(* Logix 5000 project; controller PRU vendor 1 type 14 code 107 rev 20.13; software revision 20.01; part 4 of 17 *)
(* tags used below, declared in another part *)
   AFI : BOOL;
   AlarmMaster : DINT;
   ALL_AUTO_IOK : BOOL;   // All equipment is in Auto Mode.
   ALL_DRIVES_ARE_CMD_FWD : BOOL;
   ALL_DRIVES_ARE_READY : BOOL;
   ALL_SHUTDOWN_FAULTS_IOK : BOOL;
   AUTO_FWD_CMD_GON : BOOL;
   CHANGING_TOTE_2 : BOOL;
   CHANGING_TOTE_3 : BOOL;
   CHANGING_TOTE_4 : BOOL;
   CHANGING_TOTE_5 : BOOL;
   COOLSCREW : VFD;
   DRYER : DUAL_SCREW;
   DRYER_FWD_MODE : BOOL;
   FAULTS_FA4_IOK : BOOL;   // HI TEMP FAULTS ARE OK.
   FAULTS_FA5_IOK : BOOL;
   FWD_CMD_BON : TIMER;

        [3601] := 267.2754, [3602] := 267.45117, [3603] := 267.36328, [3604] := 267.80273, [3605] := 267.71484, [3606] := 267.53906, [3607] := 267.62695, [3608] := 268.50586, [3609] := 268.41797, [3610] := 268.2422, [3611] := 268.33008, [3612] := 267.89062, [3613] := 267.97852, [3614] := 268.1543, [3615] := 268.0664, [3616] := 264.375, [3617] := 264.4629, [3618] := 264.63867, [3619] := 264.55078, [3620] := 264.99023, [3621] := 264.90234, [3622] := 264.72656, [3623] := 264.81445, [3624] := 265.69336, [3625] := 265.60547, [3626] := 265.4297, [3627] := 265.51758, [3628] := 265.07812, [3629] := 265.16602, [3630] := 265.3418, [3631] := 265.2539, [3632] := 267.0996, [3633] := 267.01172, [3634] := 266.83594, [3635] := 266.92383, [3636] := 266.48438, [3637] := 266.57227, [3638] := 266.74805, [3639] := 266.66016, [3640] := 265.78125, [3641] := 265.86914, [3642] := 266.04492, [3643] := 265.95703, [3644] := 266.39648, [3645] := 266.3086, [3646] := 266.1328, [3647] := 266.2207, [3648] := 258.75, [3649] := 258.8379, [3650] := 259.01367, [3651] := 258.92578, [3652] := 259.36523, [3653] := 259.27734, [3654] := 259.10156, [3655] := 259.18945, [3656] := 260.06836, [3657] := 259.98047, [3658] := 259.8047, [3659] := 259.89258, [3660] := 259.45312,
        [3661] := 259.54102, [3662] := 259.7168, [3663] := 259.6289, [3664] := 261.4746, [3665] := 261.38672, [3666] := 261.21094, [3667] := 261.29883, [3668] := 260.85938, [3669] := 260.94727, [3670] := 261.12305, [3671] := 261.03516, [3672] := 260.15625, [3673] := 260.24414, [3674] := 260.41992, [3675] := 260.33203, [3676] := 260.77148, [3677] := 260.6836, [3678] := 260.5078, [3679] := 260.5957, [3680] := 264.2871, [3681] := 264.19922, [3682] := 264.02344, [3683] := 264.11133, [3684] := 263.67188, [3685] := 263.75977, [3686] := 263.93555, [3687] := 263.84766, [3688] := 262.96875, [3689] := 263.05664, [3690] := 263.23242, [3691] := 263.14453, [3692] := 263.58398, [3693] := 263.4961, [3694] := 263.3203, [3695] := 263.4082, [3696] := 261.5625, [3697] := 261.6504, [3698] := 261.82617, [3699] := 261.73828, [3700] := 262.17773, [3701] := 262.08984, [3702] := 261.91406, [3703] := 262.00195, [3704] := 262.88086, [3705] := 262.79297, [3706] := 262.6172, [3707] := 262.70508, [3708] := 262.26562, [3709] := 262.35352, [3710] := 262.5293, [3711] := 262.4414, [3712] := 247.5, [3713] := 247.58789, [3714] := 247.76367, [3715] := 247.67578, [3716] := 248.11523, [3717] := 248.02734, [3718] := 247.85156, [3719] := 247.93945, [3720] := 248.81836,
        [3721] := 248.73047, [3722] := 248.55469, [3723] := 248.64258, [3724] := 248.20312, [3725] := 248.29102, [3726] := 248.4668, [3727] := 248.3789, [3728] := 250.22461, [3729] := 250.13672, [3730] := 249.96094, [3731] := 250.04883, [3732] := 249.60938, [3733] := 249.69727, [3734] := 249.87305, [3735] := 249.78516, [3736] := 248.90625, [3737] := 248.99414, [3738] := 249.16992, [3739] := 249.08203, [3740] := 249.52148, [3741] := 249.4336, [3742] := 249.25781, [3743] := 249.3457, [3744] := 253.03711, [3745] := 252.94922, [3746] := 252.77344, [3747] := 252.86133, [3748] := 252.42188, [3749] := 252.50977, [3750] := 252.68555, [3751] := 252.59766, [3752] := 251.71875, [3753] := 251.80664, [3754] := 251.98242, [3755] := 251.89453, [3756] := 252.33398, [3757] := 252.2461, [3758] := 252.07031, [3759] := 252.1582, [3760] := 250.3125, [3761] := 250.40039, [3762] := 250.57617, [3763] := 250.48828, [3764] := 250.92773, [3765] := 250.83984, [3766] := 250.66406, [3767] := 250.75195, [3768] := 251.63086, [3769] := 251.54297, [3770] := 251.36719, [3771] := 251.45508, [3772] := 251.01562, [3773] := 251.10352, [3774] := 251.2793, [3775] := 251.1914, [3776] := 258.6621, [3777] := 258.57422, [3778] := 258.39844, [3779] := 258.48633, [3780] := 258.04688,
        [3781] := 258.13477, [3782] := 258.31055, [3783] := 258.22266, [3784] := 257.34375, [3785] := 257.43164, [3786] := 257.60742, [3787] := 257.51953, [3788] := 257.95898, [3789] := 257.8711, [3790] := 257.6953, [3791] := 257.7832, [3792] := 255.9375, [3793] := 256.0254, [3794] := 256.20117, [3795] := 256.11328, [3796] := 256.55273, [3797] := 256.46484, [3798] := 256.28906, [3799] := 256.37695, [3800] := 257.25586, [3801] := 257.16797, [3802] := 256.9922, [3803] := 257.08008, [3804] := 256.64062, [3805] := 256.72852, [3806] := 256.9043, [3807] := 256.8164, [3808] := 253.125, [3809] := 253.21289, [3810] := 253.38867, [3811] := 253.30078, [3812] := 253.74023, [3813] := 253.65234, [3814] := 253.47656, [3815] := 253.56445, [3816] := 254.44336, [3817] := 254.35547, [3818] := 254.17969, [3819] := 254.26758, [3820] := 253.82812, [3821] := 253.91602, [3822] := 254.0918, [3823] := 254.0039, [3824] := 255.84961, [3825] := 255.76172, [3826] := 255.58594, [3827] := 255.67383, [3828] := 255.23438, [3829] := 255.32227, [3830] := 255.49805, [3831] := 255.41016, [3832] := 254.53125, [3833] := 254.61914, [3834] := 254.79492, [3835] := 254.70703, [3836] := 255.14648, [3837] := 255.0586, [3838] := 254.88281, [3839] := 254.9707, [3840] := 225.0,
        [3841] := 225.08789, [3842] := 225.26367, [3843] := 225.17578, [3844] := 225.61523, [3845] := 225.52734, [3846] := 225.35156, [3847] := 225.43945, [3848] := 226.31836, [3849] := 226.23047, [3850] := 226.05469, [3851] := 226.14258, [3852] := 225.70312, [3853] := 225.79102, [3854] := 225.9668, [3855] := 225.8789, [3856] := 227.72461, [3857] := 227.63672, [3858] := 227.46094, [3859] := 227.54883, [3860] := 227.10938, [3861] := 227.19727, [3862] := 227.37305, [3863] := 227.28516, [3864] := 226.40625, [3865] := 226.49414, [3866] := 226.66992, [3867] := 226.58203, [3868] := 227.02148, [3869] := 226.9336, [3870] := 226.75781, [3871] := 226.8457, [3872] := 230.53711, [3873] := 230.44922, [3874] := 230.27344, [3875] := 230.36133, [3876] := 229.92188, [3877] := 230.00977, [3878] := 230.18555, [3879] := 230.09766, [3880] := 229.21875, [3881] := 229.30664, [3882] := 229.48242, [3883] := 229.39453, [3884] := 229.83398, [3885] := 229.7461, [3886] := 229.57031, [3887] := 229.6582, [3888] := 227.8125, [3889] := 227.90039, [3890] := 228.07617, [3891] := 227.98828, [3892] := 228.42773, [3893] := 228.33984, [3894] := 228.16406, [3895] := 228.25195, [3896] := 229.13086, [3897] := 229.04297, [3898] := 228.86719, [3899] := 228.95508, [3900] := 228.51562,
        [3901] := 228.60352, [3902] := 228.7793, [3903] := 228.6914, [3904] := 236.16211, [3905] := 236.07422, [3906] := 235.89844, [3907] := 235.98633, [3908] := 235.54688, [3909] := 235.63477, [3910] := 235.81055, [3911] := 235.72266, [3912] := 234.84375, [3913] := 234.93164, [3914] := 235.10742, [3915] := 235.01953, [3916] := 235.45898, [3917] := 235.3711, [3918] := 235.19531, [3919] := 235.2832, [3920] := 233.4375, [3921] := 233.52539, [3922] := 233.70117, [3923] := 233.61328, [3924] := 234.05273, [3925] := 233.96484, [3926] := 233.78906, [3927] := 233.87695, [3928] := 234.75586, [3929] := 234.66797, [3930] := 234.49219, [3931] := 234.58008, [3932] := 234.14062, [3933] := 234.22852, [3934] := 234.4043, [3935] := 234.3164, [3936] := 230.625, [3937] := 230.71289, [3938] := 230.88867, [3939] := 230.80078, [3940] := 231.24023, [3941] := 231.15234, [3942] := 230.97656, [3943] := 231.06445, [3944] := 231.94336, [3945] := 231.85547, [3946] := 231.67969, [3947] := 231.76758, [3948] := 231.32812, [3949] := 231.41602, [3950] := 231.5918, [3951] := 231.5039, [3952] := 233.34961, [3953] := 233.26172, [3954] := 233.08594, [3955] := 233.17383, [3956] := 232.73438, [3957] := 232.82227, [3958] := 232.99805, [3959] := 232.91016, [3960] := 232.03125,
        [3961] := 232.11914, [3962] := 232.29492, [3963] := 232.20703, [3964] := 232.64648, [3965] := 232.5586, [3966] := 232.38281, [3967] := 232.4707, [3968] := 247.41211, [3969] := 247.32422, [3970] := 247.14844, [3971] := 247.23633, [3972] := 246.79688, [3973] := 246.88477, [3974] := 247.06055, [3975] := 246.97266, [3976] := 246.09375, [3977] := 246.18164, [3978] := 246.35742, [3979] := 246.26953, [3980] := 246.70898, [3981] := 246.6211, [3982] := 246.44531, [3983] := 246.5332, [3984] := 244.6875, [3985] := 244.77539, [3986] := 244.95117, [3987] := 244.86328, [3988] := 245.30273, [3989] := 245.21484, [3990] := 245.03906, [3991] := 245.12695, [3992] := 246.00586, [3993] := 245.91797, [3994] := 245.74219, [3995] := 245.83008, [3996] := 245.39062, [3997] := 245.47852, [3998] := 245.6543, [3999] := 245.5664, [4000] := 241.875, [4001] := 241.96289, [4002] := 242.13867, [4003] := 242.05078, [4004] := 242.49023, [4005] := 242.40234, [4006] := 242.22656, [4007] := 242.31445, [4008] := 243.19336, [4009] := 243.10547, [4010] := 242.92969, [4011] := 243.01758, [4012] := 242.57812, [4013] := 242.66602, [4014] := 242.8418, [4015] := 242.7539, [4016] := 244.59961, [4017] := 244.51172, [4018] := 244.33594, [4019] := 244.42383, [4020] := 243.98438,
        [4021] := 244.07227, [4022] := 244.24805, [4023] := 244.16016, [4024] := 243.28125, [4025] := 243.36914, [4026] := 243.54492, [4027] := 243.45703, [4028] := 243.89648, [4029] := 243.8086, [4030] := 243.63281, [4031] := 243.7207, [4032] := 236.25, [4033] := 236.33789, [4034] := 236.51367, [4035] := 236.42578, [4036] := 236.86523, [4037] := 236.77734, [4038] := 236.60156, [4039] := 236.68945, [4040] := 237.56836, [4041] := 237.48047, [4042] := 237.30469, [4043] := 237.39258, [4044] := 236.95312, [4045] := 237.04102, [4046] := 237.2168, [4047] := 237.1289, [4048] := 238.97461, [4049] := 238.88672, [4050] := 238.71094, [4051] := 238.79883, [4052] := 238.35938, [4053] := 238.44727, [4054] := 238.62305, [4055] := 238.53516, [4056] := 237.65625, [4057] := 237.74414, [4058] := 237.91992, [4059] := 237.83203, [4060] := 238.27148, [4061] := 238.1836, [4062] := 238.00781, [4063] := 238.0957, [4064] := 241.78711, [4065] := 241.69922, [4066] := 241.52344, [4067] := 241.61133, [4068] := 241.17188, [4069] := 241.25977, [4070] := 241.43555, [4071] := 241.34766, [4072] := 240.46875, [4073] := 240.55664, [4074] := 240.73242, [4075] := 240.64453, [4076] := 241.08398, [4077] := 240.9961, [4078] := 240.82031, [4079] := 240.9082, [4080] := 239.0625,
        [4081] := 239.15039, [4082] := 239.32617, [4083] := 239.23828, [4084] := 239.67773, [4085] := 239.58984, [4086] := 239.41406, [4087] := 239.50195, [4088] := 240.38086, [4089] := 240.29297, [4090] := 240.11719, [4091] := 240.20508, [4092] := 239.76562, [4093] := 239.85352, [4094] := 240.0293, [4095] := 239.9414);
   GTL1_PRESSURE : DINT := -395;
   GTL1_PRESSURE_Real : REAL := -19.17;
   GTL1_TEMPERATURE : DINT := 403;
   GTL2_PRESSURE : DINT := -412;
   GTL2_PRESSURE_Real : REAL := -20.34;
   GTL2_TEMPERATURE : DINT := 723;
   GTL3_PRESSURE : DINT := -355;
   GTL3_PRESSURE_Real : REAL := -21.22;
   GTL3_TEMPERATURE : DINT := 623;
   HEATER_1_ALARM_ION : BOOL := 1;
   HEATER_2_ALARM_ION : BOOL := 1;
   HEATER_3_ALARM_ION : BOOL := 1;
   HEATER_4_ALARM_ION : BOOL := 1;
   HEATER_5_ALARM_ION : BOOL := 1;
   HEATER_FAULTS_IOK : BOOL := 1;   // FA1, FA4, FA6
   HEATERS_CYCLE_ION : BOOL := 1;   // Heaters are commanded on.
   HMI_ABORT_PB : BOOL;
   HMI_Ai0_FORCE : BOOL;
   HMI_Ai0_FORCE_VALUE : REAL := 3.0;
   HMI_AI0_HI_SCALE : REAL := 100.0;
   HMI_AI0_LO_SCALE : REAL;
   HMI_Ai10_FORCE : BOOL;
   HMI_Ai10_FORCE_VALUE : REAL;
   HMI_AI10_HI_SCALE : REAL := 100.0;
   HMI_AI10_LO_SCALE : REAL;
   HMI_Ai11_FORCE : BOOL;
   HMI_Ai11_FORCE_VALUE : REAL := 33.0;
   HMI_AI11_HI_SCALE : REAL := 100.0;
   HMI_AI11_LO_SCALE : REAL;
   HMI_Ai12_FORCE : BOOL;
   HMI_Ai12_FORCE_VALUE : REAL := 42.0;
   HMI_AI12_HI_SCALE : REAL := 100.0;
   HMI_AI12_LO_SCALE : REAL;
   HMI_Ai13_FORCE : BOOL;
   HMI_Ai13_FORCE_VALUE : REAL := 35.0;
   HMI_AI13_HI_SCALE : REAL := 100.0;
   HMI_AI13_LO_SCALE : REAL;
   HMI_Ai14_FORCE : BOOL;
   HMI_Ai14_FORCE_VALUE : REAL := 42.0;
   HMI_AI14_HI_SCALE : REAL := 100.0;
   HMI_AI14_LO_SCALE : REAL;
   HMI_Ai15_FORCE : BOOL;
   HMI_Ai15_FORCE_VALUE : REAL := 37.0;
   HMI_AI15_HI_SCALE : REAL := 100.0;
   HMI_AI15_LO_SCALE : REAL;
   HMI_AI16_FORCE : BOOL;
   HMI_AI16_FORCE_VALUE : REAL := 50.0;
   HMI_AI16_HI_SCALE : REAL := 20.0;
   HMI_AI16_LO_SCALE : REAL := 4.0;
   HMI_Ai1_FORCE : BOOL;
   HMI_Ai1_FORCE_VALUE : REAL := 3.0;
   HMI_AI1_HI_SCALE : REAL := 100.0;
   HMI_AI1_LO_SCALE : REAL;
   HMI_Ai2_FORCE : BOOL;
   HMI_Ai2_FORCE_VALUE : REAL := 3.0;
   HMI_AI2_HI_SCALE : REAL := 100.0;
   HMI_AI2_LO_SCALE : REAL;
   HMI_Ai3_FORCE : BOOL;
   HMI_Ai3_FORCE_VALUE : REAL := 3.0;
   HMI_AI3_HI_SCALE : REAL := 100.0;
   HMI_AI3_LO_SCALE : REAL;
   HMI_Ai4_FORCE : BOOL;
   HMI_Ai4_FORCE_VALUE : REAL := 3.0;
   HMI_AI4_HI_SCALE : REAL := 100.0;
   HMI_AI4_LO_SCALE : REAL;
   HMI_Ai5_FORCE : BOOL;
   HMI_Ai5_FORCE_VALUE : REAL := 3.0;
   HMI_AI5_HI_SCALE : REAL := 100.0;
   HMI_AI5_LO_SCALE : REAL;
   HMI_Ai6_FORCE : BOOL;
   HMI_Ai6_FORCE_VALUE : REAL := 3.0;
   HMI_AI6_HI_SCALE : REAL := 100.0;
   HMI_AI6_LO_SCALE : REAL;
   HMI_Ai7_FORCE : BOOL;
   HMI_Ai7_FORCE_VALUE : REAL := 3.0;
   HMI_AI7_HI_SCALE : REAL := 100.0;
   HMI_AI7_LO_SCALE : REAL;
   HMI_Ai8_FORCE : BOOL;
   HMI_Ai8_FORCE_VALUE : REAL := 10.0;
   HMI_AI8_HI_SCALE : REAL := 100.0;
   HMI_AI8_LO_SCALE : REAL;
   HMI_Ai9_FORCE : BOOL;
   HMI_Ai9_FORCE_VALUE : REAL := 15.0;
   HMI_AI9_HI_SCALE : REAL := 100.0;
   HMI_AI9_LO_SCALE : REAL;
   HMI_ALARM_RESET : BOOL;
   HMI_ALARM_RESET_ONS : BOOL;
   HMI_ALARM_RESET_PB : BOOL;
   HMI_ALARM_RESET_TOF : TIMER := (PRE := 250, ACC := 256);
   HMI_ALARM_RESET_TON : TIMER := (PRE := 100);
   HMI_AUTO_SETPOINT_FDBK : REAL := 34.0;
   HMI_AUTO_START_PB : BOOL;
   HMI_CLEARING_PYROLIZER_TIME_MIN : REAL := 1.0;
   HMI_COOL_MOTOR : INT := 2;
   HMI_COOL_MOTOR_PRE : INT := 2;
   HMI_CR0_FORCE_OFF : BOOL;
   HMI_CR0_FORCE_ON : BOOL;
   HMI_CR10_FORCE_OFF : BOOL;
   HMI_CR10_FORCE_ON : BOOL;
   HMI_CR11_FORCE_OFF : BOOL;
   HMI_CR11_FORCE_ON : BOOL;
   HMI_CR12_FORCE_OFF : BOOL;
   HMI_CR12_FORCE_ON : BOOL := 1;
   HMI_CR13_FORCE_OFF : BOOL;
   HMI_CR13_FORCE_ON : BOOL;
   HMI_CR14_FORCE_OFF : BOOL;   // Knife Gate 0621 force closed.
   HMI_CR14_FORCE_ON : BOOL;   // Knife Gate 0621 force open.
   HMI_CR15_FORCE_OFF : BOOL;   // Knife Gate 0621 force closed.
   HMI_CR15_FORCE_ON : BOOL;   // Knife Gate 0621 force open.
   HMI_CR16_FORCE_OFF : BOOL;
   HMI_CR16_FORCE_ON : BOOL;
   HMI_CR17_FORCE_OFF : BOOL;
   HMI_CR17_FORCE_ON : BOOL;
   HMI_CR18_FORCE_OFF : BOOL;
   HMI_CR18_FORCE_ON : BOOL;
   HMI_CR19_FORCE_OFF : BOOL;
   HMI_CR19_FORCE_ON : BOOL;
   HMI_CR1_FORCE_OFF : BOOL;
   HMI_CR1_FORCE_ON : BOOL;
   HMI_CR2_FORCE_OFF : BOOL;
   HMI_CR2_FORCE_ON : BOOL;
   HMI_CR3_FORCE_OFF : BOOL;
   HMI_CR3_FORCE_ON : BOOL;
   HMI_CR4_FORCE_OFF : BOOL;
   HMI_CR4_FORCE_ON : BOOL;
   HMI_CR5_FORCE_OFF : BOOL;
   HMI_CR5_FORCE_ON : BOOL;
   HMI_CR6_FORCE_OFF : BOOL;
   HMI_CR6_FORCE_ON : BOOL;
   HMI_CR7_FORCE_OFF : BOOL;
   HMI_CR7_FORCE_ON : BOOL;
   HMI_CR8_FORCE_OFF : BOOL;
   HMI_CR8_FORCE_ON : BOOL;
   HMI_CR9_FORCE_OFF : BOOL;
   HMI_CR9_FORCE_ON : BOOL;
   HMI_CYCLE_0211_DELAY_TIME : DINT := 30;
   HMI_CYCLE_0221_DELAY_TIME : DINT := 30;
   HMI_CYCLE_STOP_PB_ION : BOOL;
   HMI_DCS_SPEED_FDBK : REAL := 34.0;
   HMI_DI0_FORCE_OFF : BOOL;
   HMI_DI0_FORCE_ON : BOOL;
   HMI_DI10_FORCE_OFF : BOOL;
   HMI_DI10_FORCE_ON : BOOL := 1;
   HMI_DI11_FORCE_OFF : BOOL;
   HMI_DI11_FORCE_ON : BOOL := 1;
   HMI_DI12_FORCE_OFF : BOOL;
   HMI_DI12_FORCE_ON : BOOL := 1;
   HMI_DI13_FORCE_OFF : BOOL;
   HMI_DI13_FORCE_ON : BOOL;
   HMI_DI14_FORCE_OFF : BOOL;
   HMI_DI14_FORCE_ON : BOOL;
   HMI_DI15_FORCE_OFF : BOOL;
   HMI_DI15_FORCE_ON : BOOL;
   HMI_DI16_FORCE_OFF : BOOL;
   HMI_DI16_FORCE_ON : BOOL := 1;
   HMI_DI17_FORCE_OFF : BOOL;
   HMI_DI17_FORCE_ON : BOOL := 1;
   HMI_DI18_FORCE_OFF : BOOL;
   HMI_DI18_FORCE_ON : BOOL;
   HMI_DI19_FORCE_OFF : BOOL;
   HMI_DI19_FORCE_ON : BOOL;
   HMI_DI1_FORCE_OFF : BOOL;
   HMI_DI1_FORCE_ON : BOOL;
   HMI_DI20_FORCE_OFF : BOOL;
   HMI_DI20_FORCE_ON : BOOL;
   HMI_DI21_FORCE_OFF : BOOL;
   HMI_DI21_FORCE_ON : BOOL;
   HMI_DI22_FORCE_OFF : BOOL;
   HMI_DI22_FORCE_ON : BOOL;
   HMI_DI23_FORCE_OFF : BOOL;
   HMI_DI23_FORCE_ON : BOOL;
   HMI_DI24_FORCE_OFF : BOOL;
   HMI_DI24_FORCE_ON : BOOL;
   HMI_DI25_FORCE_OFF : BOOL;
   HMI_DI25_FORCE_ON : BOOL;
   HMI_DI26_FORCE_OFF : BOOL;
   HMI_DI26_FORCE_ON : BOOL;
   HMI_DI27_FORCE_OFF : BOOL;
   HMI_DI27_FORCE_ON : BOOL;
   HMI_DI28_FORCE_OFF : BOOL;
   HMI_DI28_FORCE_ON : BOOL;
   HMI_DI29_FORCE_OFF : BOOL;
   HMI_DI29_FORCE_ON : BOOL;
   HMI_DI2_FORCE_OFF : BOOL;
   HMI_DI2_FORCE_ON : BOOL;
   HMI_DI30_FORCE_OFF : BOOL;
   HMI_DI30_FORCE_ON : BOOL;
   HMI_DI31_FORCE_OFF : BOOL;
   HMI_DI31_FORCE_ON : BOOL;
   HMI_DI3_FORCE_OFF : BOOL;
   HMI_DI3_FORCE_ON : BOOL;
   HMI_DI4_FORCE_OFF : BOOL;
   HMI_DI4_FORCE_ON : BOOL;
   HMI_DI5_FORCE_OFF : BOOL;
   HMI_DI5_FORCE_ON : BOOL;
   HMI_DI6_FORCE_OFF : BOOL;
   HMI_DI6_FORCE_ON : BOOL;
   HMI_DI7_FORCE_OFF : BOOL;
   HMI_DI7_FORCE_ON : BOOL;
   HMI_DI8_FORCE_OFF : BOOL;
   HMI_DI8_FORCE_ON : BOOL;
   HMI_DI9_FORCE_OFF : BOOL;
   HMI_DI9_FORCE_ON : BOOL := 1;
   HMI_DML_MOTOR : INT := 2;
   HMI_DML_MOTOR_PRE : INT := 2;
   HMI_DMR_MOTOR : INT := 2;
   HMI_DMR_MOTOR_PRE : INT := 2;
   HMI_DRYER_AUTO_MODE_PB : BOOL;
   HMI_DRYER_MAN_MODE_PB : BOOL;
   HMI_DRYER_OFF_MODE_PB : BOOL;
   HMI_DRYER_SEMIAUTO_MODE_PB : BOOL;
   HMI_DRYERL_SPEED : REAL := 13.470199;
   HMI_DRYERR_SPEED : REAL := 18.60265;
   HMI_DSC_SPEED_CMD : REAL := 34.0;
   HMI_FINAL_SCREW_POSITION_ERROR : REAL := -0.0030975342;
   HMI_FINISH_PROCESS_TIME_MIN : REAL := 2.0;
   HMI_HEATER_START_PB_ION : BOOL;
   HMI_HTR1_FORCED : BOOL;
   HMI_HTR1_POWER_CMD : REAL := 5.0;
   HMI_HTR2_FORCED : BOOL;
   HMI_HTR2_POWER_CMD : REAL := 5.0;
   HMI_HTR3_FORCED : BOOL;
   HMI_HTR3_POWER_CMD : REAL;
   HMI_HTR4_FORCED : BOOL;
   HMI_HTR4_POWER_CMD : REAL := 50.0;
   HMI_HTR5_FORCED : BOOL;
   HMI_HTR5_POWER_CMD : REAL;
   HMI_HTR6_FORCED : BOOL;
   HMI_HTR6_POWER_CMD : REAL := 50.0;
   HMI_HTR7_FORCED : BOOL;
   HMI_HTR7_POWER_CMD : REAL := 50.0;
   HMI_HTR8_FORCED : BOOL;
   HMI_HTR8_POWER_CMD : REAL;
   HMI_HTR9_FORCED : BOOL;
   HMI_HTR9_POWER_CMD : REAL := 50.0;
   HMI_KG021_OPEN_TIME : DINT := 30;
   HMI_KG022_OPEN_TIME : DINT := 30;
   HMI_MIX_FWD_PRESET : DINT := 400;
   HMI_MIX_REV_PRESET : DINT := -145;
   HMI_OSC_INC : REAL := 3.0;
   HMI_SEQ_1_FINAL_SETPOINT : DINT := 300;
   HMI_SEQ_1_HOLD_TIME : DINT := 90;
   HMI_SEQ_1_RATE : DINT := 3;
   HMI_SEQ_2_FINAL_SETPOINT : DINT := 600;
   HMI_SEQ_2_HOLD_TIME : DINT := 90;
   HMI_SEQ_2_RATE : DINT := 3;
   HMI_SEQ_3_FINAL_SETPOINT : DINT := 850;
   HMI_SEQ_3_HOLD_TIME : DINT := 90;
   HMI_SEQ_3_RATE : DINT := 3;
   HMI_SHUTDOWN_PB : BOOL;
   HMI_SHUTDOWN_PURGE_TIME_MIN : REAL := 1.0;
   HMI_SPARE_AO_CMD : REAL;
   HMI_SPARE_AO_FORCED : BOOL;
   HMI_STARTUP_PURGE_TIME_MIN : REAL := 0.25;
   HMI_STOP_ALL : BOOL;
   HMI_SV0201_OPEN_TIME : DINT := 5;
   HMI_SV0202_OPEN_TIME : DINT := 5;
   HMI_SYSTEM_AUTO_MODE_PB : BOOL;
   HMI_TE0101_FORCE_VALUE : INT := 2000;
   HMI_TE0101_FORCED : BOOL;
   HMI_TE0102_FORCE_VALUE : INT := 780;
   HMI_TE0102_FORCED : BOOL;
   HMI_TE0103_FORCE_VALUE : INT := 780;
   HMI_TE0103_FORCED : BOOL;
   HMI_TE0104_FORCE_VALUE : INT := 780;
   HMI_TE0104_FORCED : BOOL;
   HMI_TE0105_FORCE_VALUE : INT := 780;
   HMI_TE0105_FORCED : BOOL;
   HMI_TE0106_FORCE_VALUE : INT := 780;
   HMI_TE0106_FORCED : BOOL;
   HMI_TE0107_FORCE_VALUE : INT := 780;
   HMI_TE0107_FORCED : BOOL;
   HMI_TE0108_FORCE_VALUE : INT := 780;
   HMI_TE0108_FORCED : BOOL;
   HMI_TE0109_FORCE_VALUE : DINT := 780;
   HMI_TE0109_FORCED : BOOL;
   HMI_TE0110_FORCE_VALUE : DINT := 780;
   HMI_TE0110_FORCED : BOOL;
   HMI_TE0111_FORCE_VALUE : DINT := 780;
   HMI_TE0111_FORCED : BOOL;
   HMI_TE0112_FORCE_VALUE : DINT := 780;
   HMI_TE0112_FORCED : BOOL;
   HMI_TE0113_FORCE_VALUE : DINT := 195;
   HMI_TE0113_FORCED : BOOL;
   HMI_TE0114_FORCE_VALUE : DINT := 780;
   HMI_TE0114_FORCED : BOOL;
   HMI_TE0115_FORCE_VALUE : DINT := 780;
   HMI_TE0115_FORCED : BOOL;
   HMI_TE0116_FORCE_VALUE : DINT := 780;
   HMI_TE0116_FORCED : BOOL;
   HMI_TE0117_FORCE_VALUE : DINT := 780;
   HMI_TE0117_FORCED : BOOL;
   HMI_TE0118_FORCE_VALUE : DINT := 780;
   HMI_TE0118_FORCED : BOOL;
   HMI_TE0119_FORCE_VALUE : DINT := 780;
   HMI_TE0119_FORCED : BOOL;
   HMI_TE0120_FORCE_VALUE : DINT := 780;
   HMI_TE0120_FORCED : BOOL;
   HMI_TE0121_FORCE_VALUE : DINT := 780;
   HMI_TE0121_FORCED : BOOL;
   HMI_TE0122_FORCE_VALUE : DINT := 780;
   HMI_TE0122_FORCED : BOOL;
   HMI_TE0123_FORCE_VALUE : DINT := 780;
   HMI_TE0123_FORCED : BOOL;
   HMI_TE0124_FORCE_VALUE : DINT := 780;
   HMI_TE0124_FORCED : BOOL;
   HMI_TE0125_FORCE_VALUE : DINT := 580;
   HMI_TE0125_FORCED : BOOL;
   HMI_TE0126_FORCE_VALUE : DINT := 580;
   HMI_TE0126_FORCED : BOOL;
   HMI_TE0127_FORCE_VALUE : DINT := 580;
   HMI_TE0127_FORCED : BOOL;
   HMI_TE0128_FORCE_VALUE : DINT := 780;
   HMI_TE0128_FORCED : BOOL;
   HMI_TE0129_FORCE_VALUE : DINT := 780;
   HMI_TE0129_FORCED : BOOL;
   HMI_TE0130_FORCE_VALUE : DINT := 780;
   HMI_TE0130_FORCED : BOOL;
   HMI_TE0201_FORCE_VALUE : DINT := 100;
   HMI_TE0201_FORCED : BOOL;
   HMI_TE0202_FORCE_VALUE : DINT := 780;
   HMI_TE0202_FORCED : BOOL;
   HMI_VFD_1_JOG_FWD_PB : BOOL;
   HMI_VFD_1_JOG_REV_PB : BOOL;
   HMI_VFD_2_JOG_FWD_PB : BOOL;
   HMI_VFD_2_JOG_REV_PB : BOOL;
   HMI_WIPER_OSC_SETPOINT : REAL := 88.0;
   HMI_ZERO_SPEED_FORCE_ION : BOOL;
   HMI_ZONE1_FINAL_SETPOINT : REAL := 800.0;
   HMI_ZONE2_FINAL_SETPOINT : DINT := 1000;
   HMI_ZONE3_FINAL_SETPOINT : DINT := 1100;
   HMI_ZONE4_FINAL_SETPOINT : DINT := 850;
   HMI_ZONE5_FINAL_SETPOINT : REAL := 850.0;
   HMI_ZONE6_FINAL_SETPOINT : REAL := 1000.0;
   HMI_ZONE7_FINAL_SETPOINT : DINT := 1000;
   HMI_ZONE8_FINAL_SETPOINT : DINT := 1100;
   HMI_ZONE9_FINAL_SETPOINT : DINT := 1100;
   HTR1_CV : REAL;
   HTR1_MAX_CV_LIMIT : REAL := 100.0;
   HTR1_POWER_CMD : REAL;
   HTR2_CV : REAL;
   HTR2_MAX_CV_LIMIT : DINT := 100;
   HTR2_POWER_CMD : REAL;
   HTR3_CV : REAL := 3.2782545;
   HTR3_MAX_CV_LIMIT : REAL := 100.0;
   HTR3_POWER_CMD : REAL := 3.2781305;
   HTR4_CV : REAL;
   HTR4_MAX_CV_LIMIT : REAL := 100.0;
   HTR4_POWER_CMD : REAL;
   HTR5_CV : REAL;
   HTR5_MAX_CV_LIMIT : REAL := 100.0;
   HTR5_POWER_CMD : REAL;
   HTR6_CV : REAL;
   HTR6_MAX_CV_LIMIT : REAL := 75.0;
   HTR6_POWER_CMD : REAL;
   HTR7_CV : REAL;
   HTR7_MAX_CV_LIMIT : REAL := 100.0;
   HTR7_POWER_CMD : REAL;
   HTR8_CV : REAL := 17.512012;
   HTR8_MAX_CV_LIMIT : REAL := 100.0;
   HTR8_POWER_CMD : REAL := 17.512012;
   HTR9_CV : REAL := 22.324482;
   HTR9_MAX_CV_LIMIT : REAL := 100.0;
   HTR9_POWER_CMD : REAL := 22.324482;
   IFS_CommsLoss_TMR : TIMER := (PRE := 60000);   // Comms to IFS Has been Lost Alarm Timer
   IFS_CommsLossAlm : BOOL;   // Comms to IFS Has been Lost Alarm
   IFS_CommsWarning_TMR : TIMER := (PRE := 5000);   // Comms to IFS Has been Lost Warning Timer
   IFS_CommsWarningAlm : BOOL;   // Comms to IFS Has been Lost Warning Alarm
   IFS_PLC_Seconds_Temp : DINT := 54;
   IFS_Status_Data : PLCStatusData := (SW_Status := 11, HW_Statuts := 20, Status[0] := 2);
   IND560_Data_to_Set : SINT := 32;
   IND560_Get_Shared_Data_Message : MESSAGE;
        MessageParameters(ServiceCode := 16#000e, DestinationTag := IND560_Read_Data, ...)
   IND560_Gotton_Data : REAL;
   IND560_NetWeight : REAL;
   IND560_Read_Data : REAL := 1.1782302e-38;
   IND560_Set_Shared_Data_Message : MESSAGE;
        MessageParameters(ServiceCode := 16#0010, LocalElement := IND560_Data_to_Set, ...)
   IND560_Test_Msg : MESSAGE;
        MessageParameters(ServiceCode := 16#000e, DestinationTag := IND560_NetWeight, ...)
   INTERRUPT_INDEX : INT := 2;
   K0621_ALARM_ION : BOOL;
   K0621_IS_CLOSED : BOOL;
   K0621_IS_LOCAL : BOOL;
   K0621_IS_OPEN : BOOL := 1;
   K0621_IS_REMOTE : BOOL;
   K0622_ALARM_ION : BOOL;
   K0622_IS_CLOSED : BOOL;
   K0622_IS_LOCAL : BOOL;
   K0622_IS_OPEN : BOOL := 1;
   K0622_IS_REMOTE : BOOL;
   K6021_GO_CLOSE_GON : BOOL;
   K6021_GO_CLOSE_LON : BOOL;   // Knife Gate 6021 - Close Auto Logic
   K6021_GO_OPEN_GON : BOOL;
   K6021_GO_OPEN_LON : BOOL;   // Knife Gate 6021 - Open Auto Logic
   K6021_GO_STOP_GON : BOOL;
   K6021_GO_STOP_LON : BOOL;
   K6022_GO_CLOSE_GON : BOOL;
   K6022_GO_CLOSE_LON : BOOL;
   K6022_GO_OPEN_GON : BOOL;
   K6022_GO_OPEN_LON : BOOL;
   K6022_GO_STOP_GON : BOOL;
   K6022_GO_STOP_LON : BOOL;
   KG021_CLOSE_TON : TIMER := (PRE := 10000);
   KG021_GO_OPEN : BOOL := 1;
   KG021_MODE : INT := 3;   // 0 = OFF 1 = MAINT 2 = SEMI 3 = AUTO
   KG021_OPEN_TON : TIMER := (PRE := 10000, ACC := 10002, EN := 1, DN := 1);
   KG021_SEQ_STEP_01_DONE_TON : TIMER := (PRE := 5000);
   KG021_SEQ_STEP_02_DONE_TON : TIMER := (PRE := 5000);
   KG021_SEQ_STEP_03_DONE_TON : TIMER := (PRE := 30000);
   KG021_SEQ_STEP_04_DONE_TON : TIMER := (PRE := 30000);
   KG021_SEQUENCER : INT;   // 1 = OPEN SV0201 2 = CLOSE SV0201 3 = OPEN KG021 4 = CLOSE KG021
   KG022_CLOSE_TON : TIMER := (PRE := 10000);
   KG022_GO_OPEN : BOOL := 1;
   KG022_MODE : INT := 3;   // 0 = OFF 1 = MAINT 2 = SEMI 3 = AUTO
   KG022_OPEN_TON : TIMER := (PRE := 10000, ACC := 10003, EN := 1, DN := 1);
   KG022_SEQ_STEP_01_DONE_TON : TIMER := (PRE := 5000);
   KG022_SEQ_STEP_02_DONE_TON : TIMER := (PRE := 5000);
   KG022_SEQ_STEP_03_DONE_TON : TIMER := (PRE := 30000);
   KG022_SEQ_STEP_04_DONE_TON : TIMER := (PRE := 30000);
   KG022_SEQUENCER : INT;   // 1 = OPEN SV0202 2 = CLOSE SV0202 3 = OPEN KG022 4 = CLOSE KG022
   KPI : KPI := (PowerTotal := 24.189192, PowerPumps := 11.476128, PowerHeaters := 12.713064, EnergyTotal := 63473.797, EnergyPumps := 14235.842, EnergyHeaters := 49237.953);
   KPI_EnergyResetPB : BOOL;
   KPI_EnergyResetTmr : TIMER := (PRE := 1000);
   KPI_WeightResetPB : BOOL;
   KPI_WeightResetTmr : TIMER := (PRE := 1000);
   LEFT_AUTO_PCNT_SETPOINT : REAL := 34.0;
   LEFT_RATE : REAL := 14.501953;
   LOCAL_DATE_TIME : DateTime := (Yr := 2014, Mo := 2, Da := 4, Hr := 11, Min := 2, Sec := 52, uSec := 508603);
   LOCAL_SINE_INDEX : REAL := 6.3888044;
   LOCAL_SINE_OUTPUT : REAL := 0.10542268;
   LOCAL_TOGGLE : BOOL := 1;
   LS0211_ION : BOOL;   // KG021 OPEN LIMIT SWITCH
   LS0221_ION : BOOL;   // KG022 OPEN LIMIT SWITCH
   Major : DINT := 6;
   MASTER_RIGHT_CMD : BOOL;
   MAX_ENCODER_ERROR_MINUS : REAL := 60.63318;
   MAX_ENCODER_ERROR_MINUS_WARN : REAL := 62.63318;
   MAX_ENCODER_ERROR_PLUS : REAL := 70.63318;
   MAX_ENCODER_ERROR_PLUS_WARN : REAL := 68.63318;
   MIDNIGHT : BOOL;
   MIDNIGHT_ONS : DINT;
   Minor : DINT;
   MIX_FWD_PRESET : REAL := 400.0;
   MIX_MODE_TIMEBASE : BOOL;
   MIX_REV_PER_MIN : REAL := 1.0625;
   MIX_REV_PRESET : REAL := -145.0;
   MODE_DRYER : INT := 3;
   Module_COOL_Fault : DINT;
   Module_COOL_Iok : BOOL := 1;
   Module_COOL_Status : DINT := 16384;
   Module_DRYERL_Fault : DINT;
   Module_DRYERL_Iok : BOOL := 1;
   Module_DRYERL_Status : DINT := 16384;
   Module_DRYERR_Fault : DINT;
   Module_DRYERR_Iok : BOOL := 1;
   Module_DRYERR_Status : DINT := 16384;
   Module_ENCL_Fault : DINT;
   Module_ENCL_Iok : BOOL := 1;
   Module_ENCL_Status : DINT := 16384;
   Module_ENCR_Fault : DINT;
   Module_ENCR_Iok : BOOL := 1;
   Module_ENCR_Status : DINT := 16384;
   Module_LAI1_Fault : DINT;
   Module_LAI1_Iok : BOOL := 1;
   Module_LAI1_Status : DINT := 16384;
   Module_LAI2_Fault : DINT;
   Module_LAI2_Iok : BOOL := 1;
   Module_LAI2_Status : DINT := 16384;
   Module_LAI3_Fault : DINT;
   Module_LAI3_Iok : BOOL := 1;
   Module_LAI3_Status : DINT := 16384;
   Module_LAO1_Fault : DINT;
   Module_LAO1_Iok : BOOL := 1;
   Module_LAO1_Status : DINT := 16384;
   Module_LAO2_Fault : DINT;
   Module_LAO2_Iok : BOOL := 1;
   Module_LAO2_Status : DINT := 16384;
   Module_LDI1_Fault : DINT;
   Module_LDI1_Iok : BOOL := 1;
   Module_LDI1_Status : DINT := 16384;
   Module_LDI2_Fault : DINT;
   Module_LDI2_Iok : BOOL := 1;
   Module_LDI2_Status : DINT := 16384;
   Module_LDO1_Fault : DINT;
   Module_LDO1_Iok : BOOL := 1;
   Module_LDO1_Status : DINT := 16384;
   Module_LDO2_Fault : DINT;
   Module_LDO2_Iok : BOOL := 1;
   Module_LDO2_Status : DINT := 16384;
   Module_LTC1_Fault : DINT;
   Module_LTC1_Iok : BOOL := 1;
   Module_LTC1_Status : DINT := 16384;
   Module_LTC2_Fault : DINT;
   Module_LTC2_Iok : BOOL := 1;
   Module_LTC2_Status : DINT := 16384;
   Module_LTC3_Fault : DINT;
   Module_LTC3_Iok : BOOL := 1;
   Module_LTC3_Status : DINT := 16384;
   Module_LTC4_Fault : DINT;
   Module_LTC4_Iok : BOOL := 1;
   Module_LTC4_Status : DINT := 16384;
   MSG_ONS3 : BOOL := 1;
   myweight_2 : DINT := 45312;
   myweight_3 : DINT := 65425;
   myweight_4 : DINT := 45312;
   OK_TO_CHANGE_DIR : BOOL;
   OK_TO_STOP : BOOL;
   ONE_SEC : BOOL := 1;   // 50% Duty Cycle
   ONE_SEC_ONS : BOOL := 1;
   ONE_SEC_SS : BOOL;
   OutFeedScale : SystemAlarmMonitor;
   PF70EL_Message : MESSAGE;
        MessageParameters(ServiceCode := 16#000e, DestinationTag := VFD_1_Current, ...)
   PF70ER_Message : MESSAGE;
        MessageParameters(ServiceCode := 16#000e, DestinationTag := VFD_2_Current, ...)
   PID_1_MODE_LOCAL : BOOL;
   PID_2_MODE_LOCAL : BOOL;
   PID_3_MODE_LOCAL : BOOL;
   PID_4_MODE_LOCAL : BOOL;
   PID_5_MODE_LOCAL : BOOL;
   PID_6_MODE_LOCAL : BOOL;
   PID_7_MODE_LOCAL : BOOL;
   PID_8_MODE_LOCAL : BOOL;
   PID_9_MODE_LOCAL : BOOL;
   PID_ZONE_1 : PID := (CTL := -2147441536, EN := 1, INI := 1, OLL := 1, DVNA := 1, PVHA := 1, SP := 850.0, KP := 25.0, KI := 0.01, MAXS := 4095.0, MAXO := 100.0, UPD := 0.1, PV := 892.0, ERR := -42.0, MAXI := 4095.0, MAXCV := 100.0, MAXTIE := 4095.0, DATA[0] := 0.81552184, DATA[1] := -348.52258, DATA[2] := 892.0, DATA[3] := -42.0, DATA[4] := 850.0, DATA[5] := 0.024420025, DATA[6] := 1.0, DATA[7] := 1.6, DATA[8] := 25.0, DATA[9] := 0.01, DATA[11] := 25.0, DATA[12] := 0.01, DATA[15] := 1.0, DATA[16] := 0.024420025);
   PID_ZONE_1_MANUAL_SETPOINT : REAL := 550.0;
   PID_ZONE_1_SETPOINT : DINT := 850;
   PID_ZONE_2 : PID := (CTL := -2147441536, EN := 1, INI := 1, OLL := 1, DVNA := 1, PVHA := 1, SP := 1000.0, KP := 25.0, KI := 0.01, MAXS := 4095.0, MAXO := 100.0, UPD := 0.1, PV := 1164.75, ERR := -164.75, MAXI := 4095.0, MAXCV := 100.0, MAXTIE := 4095.0, DATA[0] := 0.5909763, DATA[1] := -455.09158, DATA[2] := 1164.75, DATA[3] := -164.75, DATA[4] := 1000.0, DATA[5] := 0.024420025, DATA[6] := 1.0, DATA[7] := 1.6, DATA[8] := 25.0, DATA[9] := 0.01, DATA[11] := 25.0, DATA[12] := 0.01, DATA[15] := 1.0, DATA[16] := 0.024420025);
   PID_ZONE_2_MANUAL_SETPOINT : REAL := 550.0;
   PID_ZONE_2_SETPOINT : DINT := 1000;
   PID_ZONE_3 : PID := (CTL := -2147449728, EN := 1, INI := 1, DVNA := 1, PVHA := 1, SP := 1100.0, KP := 25.0, KI := 0.01, MAXS := 4095.0, SO := 3.2778206, MAXO := 100.0, UPD := 0.1, PV := 1100.25, ERR := -0.25, OUT := 3.2778206, MAXI := 4095.0, MAXCV := 100.0, MAXTIE := 4095.0, DATA[0] := 3.4304457, DATA[1] := -429.8901, DATA[2] := 1100.25, DATA[3] := -0.25, DATA[4] := 1100.0, DATA[5] := 0.024420025, DATA[6] := 1.0, DATA[7] := 1.6, DATA[8] := 25.0, DATA[9] := 0.01, DATA[11] := 25.0, DATA[12] := 0.01, DATA[15] := 1.0, DATA[16] := 0.024420025);
   PID_ZONE_3_MANUAL_SETPOINT : REAL := 550.0;
   PID_ZONE_3_SETPOINT : DINT := 1100;
   PID_ZONE_4 : PID := (CTL := -2147441536, EN := 1, INI := 1, OLL := 1, DVNA := 1, PVHA := 1, SP := 850.0, KP := 30.0, KI := 0.01, MAXS := 4095.0, MAXO := 100.0, UPD := 0.1, PV := 938.0, ERR := -88.0, MAXI := 4095.0, MAXCV := 100.0, MAXTIE := 4095.0, DATA[0] := 5.1777477, DATA[1] := -366.49573, DATA[2] := 938.0, DATA[3] := -88.0, DATA[4] := 850.0, DATA[5] := 0.024420025, DATA[6] := 1.0, DATA[7] := 1.6, DATA[8] := 30.0, DATA[9] := 0.01, DATA[11] := 30.0, DATA[12] := 0.01, DATA[15] := 1.0, DATA[16] := 0.024420025);
   PID_ZONE_4_MANUAL_SETPOINT : REAL := 120.0;
   PID_ZONE_4_SETPOINT : DINT := 850;
   PID_ZONE_5 : PID := (CTL := -2147441536, EN := 1, INI := 1, OLL := 1, DVNA := 1, PVHA := 1, SP := 850.0, KP := 30.0, KI := 0.01, MAXS := 4095.0, MAXO := 100.0, UPD := 0.1, PV := 909.6667, ERR := -59.666687, MAXI := 4095.0, MAXCV := 100.0, MAXTIE := 4095.0, DATA[0] := 0.7326144, DATA[1] := -355.42532, DATA[2] := 909.6667, DATA[3] := -59.666687, DATA[4] := 850.0, DATA[5] := 0.024420025, DATA[6] := 1.0, DATA[7] := 1.6, DATA[8] := 30.0, DATA[9] := 0.01, DATA[11] := 30.0, DATA[12] := 0.01, DATA[15] := 1.0, DATA[16] := 0.024420025);
   PID_ZONE_5_MANUAL_SETPOINT : REAL := 120.0;
   PID_ZONE_5_SETPOINT : REAL := 850.0;
   PID_ZONE_6 : PID := (CTL := -2147441536, EN := 1, INI := 1, OLL := 1, DVNA := 1, PVHA := 1, SP := 1000.0, KP := 30.0, KI := 0.01, MAXS := 4095.0, MAXO := 75.0, UPD := 0.1, PV := 1103.3334, ERR := -103.333374, MAXI := 4095.0, MAXCV := 100.0, MAXTIE := 4095.0, DATA[0] := 13.186828, DATA[1] := -431.09485, DATA[2] := 1103.3334, DATA[3] := -103.333374, DATA[4] := 1000.0, DATA[5] := 0.024420025, DATA[6] := 1.0, DATA[7] := 1.6, DATA[8] := 30.0, DATA[9] := 0.01, DATA[11] := 30.0, DATA[12] := 0.01, DATA[15] := 1.0, DATA[16] := 0.024420025);
   PID_ZONE_6_MANUAL_SETPOINT : REAL := 125.0;
   PID_ZONE_6_SETPOINT : REAL := 1000.0;
   PID_ZONE_7 : PID := (CTL := -2147441536, EN := 1, INI := 1, OLL := 1, DVNA := 1, PVHA := 1, SP := 1000.0, KP := 30.0, KI := 0.01, MAXS := 4095.0, MAXO := 100.0, UPD := 0.1, PV := 1085.3334, ERR := -85.333374, MAXI := 4095.0, MAXCV := 100.0, MAXTIE := 4095.0, DATA[0] := 19.283415, DATA[1] := -424.0619, DATA[2] := 1085.3334, DATA[3] := -85.333374, DATA[4] := 1000.0, DATA[5] := 0.024420025, DATA[6] := 1.0, DATA[7] := 1.6, DATA[8] := 30.0, DATA[9] := 0.01, DATA[11] := 30.0, DATA[12] := 0.01, DATA[15] := 1.0, DATA[16] := 0.024420025);
   PID_ZONE_7_MANUAL_SETPOINT : REAL := 127.0;
   PID_ZONE_7_SETPOINT : DINT := 1000;
   PID_ZONE_8 : PID := (CTL := -2147449216, EN := 1, INI := 1, DVNA := 1, DVPA := 1, PVHA := 1, SP := 1100.0, KP := 30.0, KI := 0.01, MAXS := 4095.0, SO := 17.512012, MAXO := 100.0, UPD := 0.1, PV := 1100.0, OUT := 17.512012, MAXI := 4095.0, MAXCV := 100.0, MAXTIE := 4095.0, DATA[0] := 17.512012, DATA[1] := -429.79245, DATA[2] := 1100.0, DATA[4] := 1100.0, DATA[5] := 0.024420025, DATA[6] := 1.0, DATA[7] := 1.6, DATA[8] := 30.0, DATA[9] := 0.01, DATA[11] := 30.0, DATA[12] := 0.01, DATA[15] := 1.0, DATA[16] := 0.024420025);
   PID_ZONE_8_MANUAL_SETPOINT : REAL := 128.0;
   PID_ZONE_8_SETPOINT : DINT := 1100;
   PID_ZONE_9 : PID := (CTL := -2147449216, EN := 1, INI := 1, DVNA := 1, DVPA := 1, PVHA := 1, SP := 1100.0, KP := 30.0, KI := 0.01, MAXS := 4095.0, SO := 22.324482, MAXO := 100.0, UPD := 0.1, PV := 1100.0, OUT := 22.324482, MAXI := 4095.0, MAXCV := 100.0, MAXTIE := 4095.0, DATA[0] := 22.324482, DATA[1] := -429.79245, DATA[2] := 1100.0, DATA[4] := 1100.0, DATA[5] := 0.024420025, DATA[6] := 1.0, DATA[7] := 1.6, DATA[8] := 30.0, DATA[9] := 0.01, DATA[11] := 30.0, DATA[12] := 0.01, DATA[15] := 1.0, DATA[16] := 0.024420025);
   PID_ZONE_9_MANUAL_SETPOINT : REAL := 129.0;
   PID_ZONE_9_SETPOINT : DINT := 1100;
   PLC_Time : DINT[8] := ([0] := 2014, [1] := 2, [2] := 4, [3] := 11, [4] := 2, [5] := 50, [6] := 709640);
   PROCESS_SEQUENCER : INT := 7;
   PROCESSOR_FAULT : BOOL;
   PRODUCTION_ION : BOOL := 1;
   PRU_ShotEnabledTestTmr : TIMER := (PRE := 99999999, ACC := 14319, EN := 1, TT := 1);
   PRU_ShotEnabledTestTmrONS : BOOL;
   PRU_Status_Data : PLCStatusData := (PLCSenonds := 50, CommsWarnSecSP := 5, CommsLossSecSP := 60, Status[0] := 1298, Status[1] := 3998, Status[7] := 403, Status[8] := 723, Status[9] := 623); {produced}
        .ALARMMASTER.0   // AlarmMaster Message
        .ALARMMASTER.1   // AlarmMaster Warning
        .ALARMMASTER.2   // CSS Start Disable
        .ALARMMASTER.3   // PRU Start Disable
        .ALARMMASTER.4   // PRU Run Disable
        .STATUS[0]   // IFS Shot Time Seconds
        .STATUS[1]   // IFS Total Mix Time Seconds
        .STATUS[2]   // IFS Command Bits
        .STATUS[2].0   // IFS Run Enable
        .STATUS[2].1   // MIX_MODE_TIMEBASE 0=Mix Mode 1=Continuous Mode
   PS0101_ION : BOOL := 1;   // PRESSURE SWITCH - CONTROL PANEL Y/Z N2 PURGE
   PS0102_ION : BOOL := 1;   // PRESSURE SWITCH - MAIN N2 SUPPLY
   PVTIME_OSC_1 : TIMER := (PRE := 36000, ACC := 29417, EN := 1, TT := 1);
   PVTIME_OSC_2 : TIMER := (PRE := 2000);
   PVTIME_UPDATE : BOOL;
   PYRO_CYCLE_TIME_RESET_ONS : BOOL := 1;
   PYRO_CYCLE_TIME_RESET_SS : BOOL;
   PYRO_FWD_RUN_IOK : BOOL := 1;
   PYRO_FWD_TON : TIMER := (PRE := 2000, ACC := 2000, EN := 1, DN := 1);
   RAMP_COUNT : DINT := 55;
   RAMP_TIME : DINT := 200;
   RAMPING_SPEED_DOWN : BOOL := 1;
   RAMPING_SPEED_UP : BOOL;
   RelaxEncoderFaultTime_SpeedSP : REAL := 10.0;
   RelaxEncoderFaultTime_SpeedSP_Rev : REAL := -10.0;
   REQUEST_TO_STOP : BOOL;   // HMI MIXING SCREEN - REQUEST TO STOP WHEN SCREWS ARE NEAR ZERO.
   REQUEST_TO_STOP_L : BOOL;
   RESUME_DISCHARGE : BOOL;
   RETENTION_TIME_MIN : REAL := 50.82353;
   REV_CMD_BON : TIMER := (PRE := 1500);
   Revision : DINT := 3;
   RIGHT_AUTO_PCNT_SETPOINT : REAL := 34.02633;
   RIGHT_RATE : REAL := 14.941406;
   SCREW_ENCODERS : SCREW_ENCODERS := (GS_LEFT_ENCODER_INT_IN := 3482, GS_RIGHT_ENCODER_INT_IN := 1536, LEFT_ENCODER_DEG_OUT_REAL_OUT := 204.16992, RIGHT_ENCODER_DEG_OUT_REAL_OUT := 270.0, LEFT_RIGHT_ENCODER_ERROR_DEG_REAL_OUT := 65.63008, LEFT_ENCODER_DEG_WAS_SCANRATE_MOVED_OUT := -18.457031, RIGHT_ENCODER_DEG_WAS_SCANRATE_MOVED_OUT := -18.457031, ENCODER_MOVED_LAST_SEC_REAL_OUT := -18.457031, MIX_REV_PER_MIN_REAL_OUT := 1.0625, RETENTION_TIME_MIN_REAL_OUT := 50.82353, MIX_FWD_PRESET_REAL_IN := 400.0, MIX_REV_PRESET_REAL_IN := -145.0, ENCODER_ACC_REAL_OUT := -49.48242, SREW_MODE_INT_IN := 3, SCREW_PITCH_CONSTANT_REAL_IN := 54.0, ENCODER_OFFSET_IN := -0.2);
   SCREW_PITCH_CONSTANT : REAL := 54.0;
   SCREW_SPEED : SCREW_SPEED := (IN_SCREW_MODE := 3, IN_AUTO_FWD_CMD_BOOL := 1, IN_DCS_AUTO_SCREW_CMD_PCNT := 34.0, OUT_DCS_MASTER_SPEED_CMD := 34.0, IN_HMI_SEMIAUTO_SCREW_CMD_PCNT := 34.0, OUT_MASTER_AUTO_SETPOINT_PCNT := 34.0, IN_LEFT_RIGHT_ENCODER_ERROR_DEG := 65.63008, IN_WIPER_OSC_SETPOINT := 65.63318, OUT_FINAL_SCREW_POSITION_ERROR := -0.0030975342, OUT_AUTO_SCREW_LEFT_CMD_FREQ := 5145.56, OUT_AUTO_SCREW_RIGHT_CMD_FREQ := 5149.5444, IN_LEFT_VFD_ION := 1, IN_RIGHT_VFD_ION := 1, IN_LEFT_VFD_ACTUAL := 1, IN_RIGHT_VFD_ACTUAL := 1, IN_SCREW_FAULTED_IOK := 1, OUT_LEFT_AUTO_PCNT_SETPOINT := 34.0, OUT_RIGHT_AUTO_PCNT_SETPOINT := 34.02633, IN_LEFT_VFD_ACTUAL_FREQ := 799, IN_RIGHT_VFD_ACTUAL_FREQ := 719, OUT_LEFT_VFD_ACTUAL_SPEED_PERCENT := 5.2795033, OUT_RIGHT_VFD_ACTUAL_SPEED_PERCENT := 4.750892, CALC_COMP_LIMIT := 17.0);
   SCREW_SPEED_OUT_L : REAL := 5145.56;
   SCREW_SPEED_OUT_R : REAL := 5149.5444;
   SCREW_WIPE : SCREW_WIPER := (HMI_WIPE_INC_REAL_IN := 3.0, HMI_WIPE_SETPOINT_REAL_IN := 88.0, WIPE_HOLD_TIME_DINT_IN := 90, WIPER_OSC_REAL_OUT := 65.63318, WIPE_EON_IN := 1, WIPE_FREEZE_IN := 1);
   SCREWS_ENABLE_GON : BOOL := 1;   // Dryer screw faults are ok.
   SCREWS_WIPE_HOLD_TIME : DINT := 90;
   SEQ_1_HOLD_REM : REAL := 5400000.0;
   SEQ_1_HOLD_REM_MIN : REAL := 90.0;
   SEQ_1_HOLD_TIME : DINT := 5400000;
   SEQ_1_HOLD_TON : TIMER := (PRE := 5400000);
   SEQ_1_HOLDING_ION : BOOL;
   SEQ_1_ION : BOOL;
   SEQ_2_HOLD_REM : REAL := 5400000.0;
   SEQ_2_HOLD_REM_MIN : REAL := 90.0;
   SEQ_2_HOLD_TIME : DINT := 5400000;
   SEQ_2_HOLD_TON : TIMER := (PRE := 5400000);
   SEQ_2_HOLDING_ION : BOOL;
   SEQ_2_ION : BOOL;
   SEQ_3_HOLD_REM : REAL := 5400000.0;
   SEQ_3_HOLD_REM_MIN : REAL := 90.0;
   SEQ_3_HOLD_TIME : DINT := 5400000;
   SEQ_3_HOLD_TON : TIMER := (PRE := 5400000);
   SEQ_3_HOLDING_ION : BOOL;
   SEQ_3_ION : BOOL;
   SEQ_RATE : REAL;
   SEQ_SHUTDOWN_ONS : BOOL;
   SEQ_STEP_00_DONE_TON : TIMER;
   SEQ_STEP_00_DONEA : BOOL := 1;   // ALL_AUTO_IOK
   SEQ_STEP_00_DONEB : BOOL := 1;   // ALL_DRIVES_ARE_READY
   SEQ_STEP_00_DONEC : BOOL := 1;   // ALL_DRIVES_ARE_CMD_FWD
   SEQ_STEP_00_DONED : BOOL := 1;   // ALL_SHUTDOWN_FAULTS_IOK
   SEQ_STEP_01_DONE_TON : TIMER := (PRE := 5000);
   SEQ_STEP_01_DONEA : BOOL := 1;   // FS-0204 INDICATES FLOW IS PRESENT
   SEQ_STEP_01_DONEB : BOOL := 1;
   SEQ_STEP_01_DONEC : BOOL := 1;
   SEQ_STEP_02_DONE_TON : TIMER := (PRE := 5000);
   SEQ_STEP_02_DONEA : BOOL := 1;   // FS-0101 INDICATES FLOW IS PRESENT
   SEQ_STEP_02_DONEB : BOOL;   // TIME > HMI SP (STARTUP PURGE)
   SEQ_STEP_02_DONEC : BOOL := 1;
   SEQ_STEP_03_DONE_TON : TIMER := (PRE := 5000);
   SEQ_STEP_03_DONEA : BOOL := 1;   // HEATERS ARE ON.
   SEQ_STEP_03_DONEB : BOOL := 1;
   SEQ_STEP_03_DONEC : BOOL := 1;
   SEQ_STEP_04_DONE_TON : TIMER := (PRE := 5000);
   SEQ_STEP_04_DONEA : BOOL := 1;   // VFD0201 (ION)
   SEQ_STEP_04_DONEB : BOOL := 1;   // KG-021 (OPEN 1X)
   SEQ_STEP_04_DONEC : BOOL := 1;   // KF-022 (OPEN 1X)
   SEQ_STEP_05_DONE_TON : TIMER := (PRE := 5000);
   SEQ_STEP_05_DONEA : BOOL := 1;   // VFD0101 (ION)
   SEQ_STEP_05_DONEB : BOOL := 1;   // VFD0102 (ION)
   SEQ_STEP_05_DONEC : BOOL := 1;
   SEQ_STEP_06_DONE_TON : TIMER := (PRE := 500);
   SEQ_STEP_06_DONEA : BOOL;   // VFD0301 (ION)
   SEQ_STEP_06_DONEB : BOOL := 1;
   SEQ_STEP_06_DONEC : BOOL := 1;
   SEQ_STEP_07_DONE_TON : TIMER := (PRE := 5000);
   SEQ_STEP_07_DONEA : BOOL;
   SEQ_STEP_07_DONEB : BOOL;
   SEQ_STEP_07_DONEC : BOOL;
   SEQ_STEP_07_DONED : BOOL := 1;
   SEQ_STEP_08_DONE_TON : TIMER := (PRE := 5000);
   SEQ_STEP_08_DONEA : BOOL := 1;
   SEQ_STEP_08_DONEB : BOOL := 1;
   SEQ_STEP_08_DONEC : BOOL := 1;
   SEQ_STEP_09_DONE_TON : TIMER := (PRE := 5000);
   SEQ_STEP_09_DONEA : BOOL := 1;   // VFD0301 (IOF)
   SEQ_STEP_09_DONEB : BOOL := 1;
   SEQ_STEP_09_DONEC : BOOL := 1;
   SEQ_STEP_10_DONE_TON : TIMER := (PRE := 5000);
   SEQ_STEP_10_DONEA : BOOL;   // TIME > HMI SP (FINISH PROCESS TIME)
   SEQ_STEP_10_DONEB : BOOL := 1;
   SEQ_STEP_10_DONEC : BOOL := 1;
   SEQ_STEP_11_DONE_TON : TIMER := (PRE := 5000);
   SEQ_STEP_11_DONEA : BOOL;   // HEATERS ARE OFF.
   SEQ_STEP_11_DONEB : BOOL := 1;
   SEQ_STEP_11_DONEC : BOOL := 1;
   SEQ_STEP_12_DONE_TON : TIMER := (PRE := 5000);
   SEQ_STEP_12_DONEA : BOOL;   // TIME > HMI SP (CLEARING TIME)
   SEQ_STEP_12_DONEB : BOOL := 1;
   SEQ_STEP_12_DONEC : BOOL := 1;
   SEQ_STEP_13_DONE_TON : TIMER := (PRE := 5000);
   SEQ_STEP_13_DONEA : BOOL;   // VFD0101 (IOF)
   SEQ_STEP_13_DONEB : BOOL;   // VFD0102 (IOF)
   SEQ_STEP_13_DONEC : BOOL := 1;
   SEQ_STEP_14_DONE_TON : TIMER := (PRE := 5000);
   SEQ_STEP_14_DONEA : BOOL;   // VFD0201 (IOF)
   SEQ_STEP_14_DONEB : BOOL := 1;   // KG-021 (CLOSED)
   SEQ_STEP_14_DONEC : BOOL := 1;   // KF-022 (CLOSED)
   SEQ_STEP_15_DONE_TON : TIMER := (PRE := 5000);
   SEQ_STEP_15_DONEA : BOOL := 1;   // FS-0101 INDICATES FLOW IS PRESENT
   SEQ_STEP_15_DONEB : BOOL;   // TIME > HMI SP (SHUTDOWN PURGE)
   SEQ_STEP_15_DONEC : BOOL := 1;
   SEQ_STEP_16_DONE_TON : TIMER := (PRE := 5000);
   SEQ_STEP_16_DONEA : BOOL;   // ALL TEMPS < 200F
   SEQ_STEP_16_DONEB : BOOL := 1;
   SEQ_STEP_16_DONEC : BOOL := 1;
   SET_PYRO_SPEED_TO_ZERO : BOOL;
   SHUTDOWN_PURGE_TIME_REMAINING_SEC : REAL := 60.0;
   SHUTDOWN_PURGE_TIME_REMAINING_TEMP : REAL := 60000.0;
   SHUTDOWN_PURGE_TIMER : TIMER := (PRE := 60000);
   SLAVE_COMP_LIMIT : REAL := 17.0;
   SP_RATIO : REAL := 0.9411765;
   SPARE_AO_CMD : REAL := 50.0;
   SPEED_RAMP_FREEZE_TOF : TIMER := (PRE := 5000, EN := 1, DN := 1);
   SPEED_RAMP_MULT : REAL := 0.35;
   STANDBY_MODE_ION : BOOL;
   STANDBY_MODE_TOF : TIMER;
   STANDBY_MODE_TON : TIMER := (PRE := 10000);
   STANDBY_TEMPERATURE_SETPOINT : REAL := 900.0;
   START_ENABLE : BOOL;
   START_TOTE_CHANGE : BOOL;
   STARTUP_PURGE_TIME_REMAINING_SEC : REAL := 15.0;
   STARTUP_PURGE_TIME_REMAINING_TEMP : REAL := 15000.0;
   STARTUP_PURGE_TIMER : TIMER := (PRE := 15000);
   STEP_00_ION : BOOL;   // 0 - SYSTEM NOT OPERATING
   STEP_01_ION : BOOL;   // 1 - COOLING WATER FLOW
   STEP_02_ION : BOOL;   // 2 - STARTUP N2 PURGE
   STEP_03_ION : BOOL;   // 3 - RAMPING HEATERS TO SETPOINT
   STEP_04_ION : BOOL;   // 4 - RUNNING DISCHARGE SYSTEM
   STEP_05_ION : BOOL;   // 5 - RUNNING PYROLIZER SCREWS
   STEP_06_ION : BOOL;   // 6 - RUNNING FEED SYSTEM
   STEP_07_ION : BOOL := 1;   // 7 - SYSTEM PROCESSING
   STEP_08_ION : BOOL;   // 8 - AUTO SHUTDOWN
   STEP_09_ION : BOOL;   // 9 - STOPPING FEED SYSTEM
   STEP_10_ION : BOOL;   // 10 - FINISHING PROCESS
   STEP_11_ION : BOOL;   // 11 - STOPPING HEATERS
   STEP_12_ION : BOOL;   // 12 - CLEARING PYROLIZER
   STEP_13_ION : BOOL;   // 13 - STOPPING PYROLIZER
   STEP_14_ION : BOOL;   // 14 - STOPPING DISCHARGE SYSTEM
   STEP_15_ION : BOOL;   // 15 - SHUTDOWN N2 PURGE
   STEP_16_ION : BOOL;   // 16 - WAITING FOR SYSTEM COOL
   SV0101 : BOOL;
   SV0101_LON : BOOL;
   SV0102 : BOOL := 1;
   SV0102_LON : BOOL := 1;
   SV0201 : BOOL;
   SV0201_LON : BOOL;
   SV0202 : BOOL := 1;
   SV0202_LON : BOOL;
   SV0203 : BOOL := 1;
   SV0203_LON : BOOL := 1;
   SYSTEM_SETPOINT : REAL := 800.0;
   TE0101 : REAL := 894.0;
   TE0101_RAW : DINT := 894;
   TE0101_SEL_ION : BOOL := 1;
   TE0102 : REAL := 890.0;
   TE0102_RAW : DINT := 890;
   TE0102_SEL_ION : BOOL := 1;
   TE0103 : REAL := 895.0;
   TE0103_RAW : DINT := 895;
   TE0103_SEL_ION : BOOL := 1;
   TE0104 : REAL := 889.0;
   TE0104_RAW : DINT := 889;
   TE0104_SEL_ION : BOOL := 1;
   TE0105 : REAL := 1171.0;
   TE0105_RAW : DINT := 1171;
   TE0105_SEL_ION : BOOL := 1;
   TE0106 : REAL := 1168.0;
   TE0106_RAW : DINT := 1168;
   TE0106_SEL_ION : BOOL := 1;
   TE0107 : REAL := 1164.0;
   TE0107_RAW : DINT := 1164;
   TE0107_SEL_ION : BOOL := 1;
   TE0108 : REAL := 1156.0;
   TE0108_RAW : DINT := 1156;
   TE0108_SEL_ION : BOOL := 1;
   TE0109 : REAL := 1113.0;
   TE0109_RAW : DINT := 1113;
   TE0109_SEL_ION : BOOL := 1;
   TE0110 : REAL := 1108.0;
   TE0110_RAW : DINT := 1108;
   TE0110_SEL_ION : BOOL := 1;
   TE0111 : REAL := 1099.0;
   TE0111_RAW : DINT := 1099;
   TE0111_SEL_ION : BOOL := 1;
   TE0112 : REAL := 1081.0;
   TE0112_RAW : DINT := 1081;
   TE0112_SEL_ION : BOOL := 1;
   TE0113 : REAL := 939.0;
   TE0113_RAW : DINT := 939;
   TE0113_SEL_ION : BOOL := 1;
   TE0114 : REAL := 923.0;
   TE0114_RAW : DINT := 923;
   TE0114_SEL_ION : BOOL := 1;
   TE0115 : REAL := 912.0;
   TE0115_RAW : DINT := 912;
   TE0115_SEL_ION : BOOL := 1;
   TE0116 : REAL := 895.0;
   TE0116_RAW : DINT := 895;
   TE0116_SEL_ION : BOOL := 1;
   TE0117 : REAL := 1124.0;
   TE0117_RAW : DINT := 1124;
   TE0117_SEL_ION : BOOL := 1;
   TE0118 : REAL := 1090.0;
   TE0118_RAW : DINT := 1090;
   TE0118_SEL_ION : BOOL := 1;
   TE0119 : REAL := 1076.0;
   TE0119_RAW : DINT := 1076;
   TE0119_SEL_ION : BOOL := 1;
   TE0120 : REAL := 1093.0;
   TE0120_RAW : DINT := 1093;
   TE0120_SEL_ION : BOOL := 1;
   TE0121 : REAL := 1101.0;
   TE0121_RAW : DINT := 1101;
   TE0121_SEL_ION : BOOL := 1;
   TE0122 : REAL := 1107.0;
   TE0122_RAW : DINT := 1107;
   TE0122_SEL_ION : BOOL := 1;
   TE0123 : REAL := 1104.0;
   TE0123_RAW : DINT := 1104;
   TE0123_SEL_ION : BOOL := 1;
   TE0124 : REAL := 1093.0;
   TE0124_RAW : DINT := 1093;
   TE0124_SEL_ION : BOOL := 1;
   TE0125 : REAL := 952.0;
   TE0125_RAW : DINT := 952;
   TE0125_SEL_ION : BOOL := 1;
   TE0126 : REAL := 922.0;
   TE0126_RAW : DINT := 922;
   TE0126_SEL_ION : BOOL := 1;
   TE0127 : REAL := 1096.0;
   TE0127_RAW : DINT := 1096;
   TE0127_SEL_ION : BOOL := 1;
   TE0128 : REAL := 1087.0;
   TE0128_RAW : DINT := 1087;
   TE0128_SEL_ION : BOOL := 1;
   TE0129 : REAL := 1092.0;
   TE0129_RAW : DINT := 1092;
   TE0129_SEL_ION : BOOL := 1;
   TE0130 : REAL := 1103.0;
   TE0130_RAW : DINT := 1103;
   TE0130_SEL_ION : BOOL := 1;
   TE0201 : REAL := 118.0;
   TE0201_RAW : DINT := 118;
   TE0202 : REAL := 99.0;
   TE0202_RAW : DINT := 99;
   TEMP_ZONE_1_AVE : REAL;
   TempDint : DINT := 65428;
   TEMPERATURE_SETPOINT_IS_RAMPING : BOOL;
   TEST_HTR1_CV_LIMIT : BOOL := 1;
   TEST_HTR2_CV_LIMIT : BOOL := 1;
   TEST_HTR3_CV_LIMIT : BOOL := 1;
   TEST_HTR4_CV_LIMIT : BOOL := 1;
   TEST_HTR5_CV_LIMIT : BOOL := 1;
   TEST_HTR6_CV_LIMIT : BOOL := 1;
   TEST_HTR7_CV_LIMIT : BOOL := 1;
   TEST_HTR8_CV_LIMIT : BOOL := 1;
   TEST_HTR9_CV_LIMIT : BOOL := 1;
   TEST_INDEX : INT := 5000;
   TEST_KG021 : BOOL;
   TEST_KG022 : BOOL;
   TEST_VFD_BON : BOOL := 1;
   testdint : DINT := -1342177154;
   testjpm : BOOL := 1;
   THRESHOLD : REAL[9000] := ([404] := 3.0, [500] := 12.5, [501] := 12.5, [600] := 1375.0, [601] := 1375.0, [602] := 1375.0, [603] := 1375.0, [604] := 1375.0, [605] := 1375.0, [606] := 1375.0, [607] := 1375.0, [608] := 1375.0, [609] := 1375.0, [610] := 1375.0, [611] := 1375.0, [612] := 1375.0, [613] := 1375.0, [614] := 1375.0, [615] := 1375.0, [616] := 1375.0, [617] := 1375.0, [618] := 1375.0, [619] := 1375.0, [620] := 1375.0, [621] := 1375.0, [622] := 1375.0, [623] := 1375.0, [624] := 1375.0, [625] := 1375.0, [626] := 1375.0, [627] := 1375.0, [628] := 1375.0, [629] := 1375.0, [630] := 1375.0, [631] := 1375.0, [800] := 1200.0, [801] := 1400.0, [3006] := 13.65, [3016] := 13.0, [3017] := 0.3, [3021] := 13.65, [3112] := 20.0, [4000] := 1550.0, [4001] := 1550.0, [4002] := 1550.0, [4003] := 1550.0, [4004] := 1550.0, [4005] := 1550.0, [4006] := 1550.0, [4007] := 1550.0, [4008] := 1550.0, [4009] := 1550.0, [4010] := 1550.0, [4011] := 1550.0, [4012] := 1475.0, [4013] := 1475.0, [4014] := 1475.0, [4015] := 1475.0, [4016] := 1475.0, [4017] := 1475.0,
        [4018] := 1475.0, [4019] := 1475.0, [4020] := 1475.0, [4021] := 1475.0, [4022] := 1475.0, [4023] := 1475.0, [4024] := 1475.0, [4025] := 1475.0, [4026] := 1475.0, [4027] := 1475.0, [4028] := 1475.0, [4029] := 1475.0, [4030] := 1475.0, [4031] := 1475.0, [4100] := 1000.0, [4200] := 1000.0, [5006] := 5.0, [5008] := 1.0, [5016] := 3.2, [5805] := 100.0, [5806] := 100.0, [5807] := 100.0, [5808] := 60.0, [5809] := 60.0, [5810] := 60.0, [5811] := 60.0, [5812] := 60.0, [5813] := 60.0, [5814] := 60.0, [5815] := 60.0, [5816] := 60.0, [5817] := 60.0, [5818] := 60.0, [5819] := 60.0);
   TIMER_MSG_OFF : TIMER := (PRE := 250, ACC := 11, EN := 1, TT := 1);
   TIMER_MSG_ON : TIMER := (PRE := 250, ACC := 46, EN := 1, TT := 1);
   TIMER_ONE_SEC_OFF : TIMER := (PRE := 500, ACC := 503, EN := 1, DN := 1);
   TIMER_ONE_SEC_ON : TIMER := (PRE := 500, ACC := 261, EN := 1, TT := 1);
   TIMER_WDT_OFF : TIMER := (PRE := 1500, ACC := 1504, EN := 1, DN := 1);
   TIMER_WDT_ON : TIMER := (PRE := 1500, ACC := 755, EN := 1, TT := 1);
   TOTAL_SCAN_COUNT : DINT := 3998;
   TOTAL_SCAN_COUNTING : DINT := 2365;
   TOTAL_SCAN_SEC : REAL := 39.98;
   TOTE_CHANGE_MODE : INT;
   TOTE_CHANGE_REMAINING : REAL;
   TOTE_CHANGE_REMAINING_MS : REAL := 600000.0;
   TOTE_CHANGE_SETPOINT : DINT := 10;
   TOTE_CHANGE_TIMED_OUT : BOOL;
   TOTE_CHANGEOUT_TOF : TIMER := (PRE := 20000, ACC := 20004, EN := 1, DN := 1);
   TOTE_CHANGEOUT_TON : TIMER := (PRE := 1800000);
   TOTE_WEIGHT : REAL := -5.0;
   UTL_CommsLoss_TMR : TIMER := (PRE := 60000, EN := 1, TT := 1);   // Comms to UTL Has been Lost Alarm Timer
   UTL_CommsLossAlm : BOOL;   // Comms to UTL Has been Lost Alarm
   UTL_CommsWarning_TMR : TIMER := (PRE := 5000, EN := 1, TT := 1);   // Comms to UTL Has been Lost Warning Timer
   UTL_CommsWarningAlm : BOOL;   // Comms to UTL Has been Lost Warning Alarm
   UTL_PLC_Seconds_Temp : DINT := 50;
   UTL_Status_Data : PLCStatusData := (PLCSenonds := 51, AlarmMaster := 3, CommsWarnSecSP := 5, CommsLossSecSP := 60, OptionH3 := 1, Status[0] := 3, Status[9] := 9999);
        .STATUS[0].2   // CRITICAL Loss of House Power
   VAPOR_1 : REAL := -1.11;
   VAPOR_1_TEMP : DINT := 100;
   VAPOR_2 : REAL := -1.22;
   VAPOR_2_TEMP : DINT := 200;
   VAPOR_3 : REAL := -1.33;
   VAPOR_3_TEMP : DINT := 300;
   VFD_1_Current : DINT := 610;
   VFD_1_Current_Real : REAL := 6.1;
   VFD_1_Tot : EnergyTot := (EI := 5.1, Power := 4.48416, Energy := 6183.0303, kWh_Tmr.PRE := 1000, kWh_Tmr.EN := 1, kWh_Tmr.TT := 1, kWh_SampleTime := 1.0, kWh_TimeMultiplier := 3600.0);   // Left Dryer
   VFD_2_Current : DINT := 660;
   VFD_2_Current_Real : REAL := 6.8;
   VFD_2_Tot : EnergyTot := (EI := 6.1, Power := 5.3976, Energy := 6322.6606, kWh_Tmr.PRE := 1000, kWh_Tmr.EN := 1, kWh_Tmr.TT := 1, kWh_SampleTime := 1.0, kWh_TimeMultiplier := 3600.0);   // Right Dryer
   VFD_3_Current : DINT := 192;
   VFD_3_Current_Real : REAL := 1.92;
   VFD_3_Tot : EnergyTot := (EI := 1.92, Power := 1.5943679, Energy := 1730.1501, kWh_Tmr.PRE := 1000, kWh_SampleTime := 1.0, kWh_TimeMultiplier := 3600.0);   // Cooling Screw
   VFD_AUTO_RESET : BOOL;
   VFD_CommsFaultTest : DINT := 1755;
   VFD_COOLSCREW_CONTROL : VFD_Motor_Control := (IN_HARD_STOP := 1, IN_RUN_INTERLOCK_1 := 1, IN_RUN_INTERLOCK_2 := 1, IN_RUN_INTERLOCK_3 := 1, IN_VFD_IS_READY := 1, IN_CURRENT_PROCESS_SEQUENCER_STEP := 7, IN_PROCESS_SEQUENCER_AUTO_START_STEP := 4, IN_PROCESS_SEQUENCER_AUTO_STOP_STEP := 13, IN_HMI_SEMI_SPEED_SETPOINT_PCNT := 40.0, IN_AUTO_SPEED_SETPOINT_PERCENT := 40.0, IN_VFD_SPEED_SCALE := 6.0, IN_VFD_ACTUAL_FREQ := 240.0, IN_VFD_IS_RUNNING := 1, OUT_AUTO_MODE_ION := 1, OUT_MODE := 3, OUT_FWD_COMMAND := 1, OUT_VFD_RUN_COMMAND := 1, OUT_CMD_RUN_ENABLED := 1, OUT_START_CMD_AUTO := 1, OUT_VFD_SPEED_SETPOINT_COMMAND := 240, OUT_VFD_ACTUAL_SPEED_PERCENT := 40.0, OUT_RUNNING_BON := 1);
   VFD_SHUTDOWN_TEMP : DINT := 230;
   VFDS_BON : BOOL := 1;   // DRYER VFDs HAVE BEEN COMMANDED ON FOR 1 SECOND.
   VFDS_TON : TIMER := (PRE := 1000, ACC := 1000, EN := 1, DN := 1);
   WARNA_IOK : BOOL := 1;
   WARNB_IOK : BOOL := 1;
   WARNC_IOK : BOOL := 1;
   WARND_IOK : BOOL := 1;
   WARNE_IOK : BOOL := 1;
   WARNF_IOK : BOOL := 1;
   WARNG_IOK : BOOL := 1;
   WARNING_FAULTS_IOK : BOOL := 1;
   WC025_DailyResetPB : BOOL;
   WC025_DailyTotal : REAL := 3323.0;
   WC025_DailyTotalLast : REAL;
   WC025_DailyTotalResetPB_ONS : BOOL := 1;
   WC025_TareALM : BOOL := 1;
   WDT_ONS : BOOL := 1;
   WDT_SS : BOOL;
   WEIGHT : REAL;
   WIPE_ACTUAL : REAL := 65.63318;
   WIPE_EON : BOOL := 1;
   WIPE_FREEZE_CMD : BOOL := 1;
   WIPE_HOLDING : BOOL;
   WIPE_MASTER : BOOL;
   WIPE_MASTER_BOF : TIMER := (PRE := 10000, ACC := 10000, EN := 1, DN := 1);
   WIPE_MASTER_BON : TIMER := (PRE := 10000);
   WIPE_MASTER_ONS : BOOL := 1;
   WIPE_MASTER_SS : BOOL;
   WIPE_PERIOD_COUNTS_ACC : REAL := 4779.0;
   WIPE_PERIOD_ONS : BOOL := 1;
   WIPE_PERIOD_SECONDS : REAL := 581.04;
   WIPE_TON : TIMER := (PRE := 10000, ACC := 10000, EN := 1, DN := 1);
   Z1_AMPS_TEMP : REAL := 0.16;
   Z1_L1_AMPS : REAL := 0.06;
   Z1_L2_AMPS : REAL := 0.099999994;
   Z1_L3_AMPS : REAL := 0.11;
   Z1L1_Tot : EnergyTot := (EI := 0.06, Power := 0.016647398, Energy := 4723.5303, kWh_Tmr.PRE := 1000, kWh_SampleTime := 1.0, kWh_TimeMultiplier := 3600.0);
   Z1L2_Tot : EnergyTot := (EI := 0.099999994, Power := 0.027745662, Energy := 4578.37, kWh_Tmr.PRE := 1000, kWh_SampleTime := 1.0, kWh_TimeMultiplier := 3600.0);
   Z1L3_Tot : EnergyTot := (EI := 0.11, Power := 0.03052023, Energy := 4568.22, kWh_Tmr.PRE := 1000, kWh_Tmr.EN := 1, kWh_Tmr.TT := 1, kWh_SampleTime := 1.0, kWh_TimeMultiplier := 3600.0);
   Z2_AMPS_TEMP : REAL := 0.12;
   Z2_L1_AMPS : REAL := 0.06;
   Z2_L2_AMPS : REAL := 0.06;
   Z2_L3_AMPS : REAL := 0.02;
   Z2L1_Tot : EnergyTot := (EI := 0.06, Power := 0.019421965, Energy := 2626.3103, kWh_Tmr.PRE := 1000, kWh_SampleTime := 1.0, kWh_TimeMultiplier := 3600.0);
   Z2L2_Tot : EnergyTot := (EI := 0.06, Power := 0.016647398, Energy := 2607.7402, kWh_Tmr.PRE := 1000, kWh_SampleTime := 1.0, kWh_TimeMultiplier := 3600.0);
   Z2L3_Tot : EnergyTot := (EI := 0.02, Power := 0.0055491324, Energy := 2612.5403, kWh_Tmr.PRE := 1000, kWh_SampleTime := 1.0, kWh_TimeMultiplier := 3600.0);
   Z3_AMPS_TEMP : REAL := 4.76;
   Z3_L1_AMPS : REAL := 2.4199998;
   Z3_L2_AMPS : REAL := 2.32;
   Z3_L3_AMPS : REAL := 1.9799999;
   Z3L1_Tot : EnergyTot := (EI := 2.77, Power := 0.6131792, Energy := 1917.4602, kWh_Tmr.PRE := 1000, kWh_Tmr.EN := 1, kWh_Tmr.TT := 1, kWh_SampleTime := 1.0, kWh_TimeMultiplier := 3600.0);
   Z3L2_Tot : EnergyTot := (EI := 3.1899998, Power := 0.5604624, Energy := 1975.5702, kWh_Tmr.PRE := 1000, kWh_Tmr.EN := 1, kWh_Tmr.TT := 1, kWh_SampleTime := 1.0, kWh_TimeMultiplier := 3600.0);
   Z3L3_Tot : EnergyTot := (EI := 2.79, Power := 0.59930634, Energy := 1971.4001, kWh_Tmr.PRE := 1000, kWh_Tmr.ACC := 1000, kWh_Tmr.EN := 1, kWh_Tmr.DN := 1, kWh_SampleTime := 1.0, kWh_TimeMultiplier := 3600.0);
   Z4_L1_AMPS : REAL := 0.01;
   Z4L1_Tot : EnergyTot := (EI := 0.01, Power := 0.0027745662, Energy := 3143.2202, kWh_Tmr.PRE := 1000, kWh_SampleTime := 1.0, kWh_TimeMultiplier := 3600.0);
   Z5_L2_AMPS : REAL := 0.08;
   Z5L2_Tot : EnergyTot := (EI := 0.08, Power := 0.02219653, Energy := 5744.0503, kWh_Tmr.PRE := 1000, kWh_SampleTime := 1.0, kWh_TimeMultiplier := 3600.0);
   Z6_L3_AMPS : REAL := 0.01;
   Z6L3_Tot : EnergyTot := (EI := 0.02, Power := 0.0027745662, Energy := 1042.6101, kWh_Tmr.PRE := 1000, kWh_SampleTime := 1.0, kWh_TimeMultiplier := 3600.0);
   Z7_L1_AMPS : REAL := 0.089999996;
   Z7L1_Tot : EnergyTot := (EI := 0.089999996, Power := 0.024971096, Energy := 3900.8103, kWh_Tmr.PRE := 1000, kWh_SampleTime := 1.0, kWh_TimeMultiplier := 3600.0);
   Z8_L2_AMPS : REAL := 18.27;
   Z8L2_Tot : EnergyTot := (EI := 18.699999, Power := 5.041387, Energy := 3364.3503, kWh_Tmr.PRE := 1000, kWh_Tmr.ACC := 1000, kWh_Tmr.EN := 1, kWh_Tmr.DN := 1, kWh_SampleTime := 1.0, kWh_TimeMultiplier := 3600.0);
   Z9_L3_AMPS : REAL := 19.529999;
   Z9L3_Tot : EnergyTot := (EI := 19.529999, Power := 5.3410406, Energy := 4461.7803, kWh_Tmr.PRE := 1000, kWh_SampleTime := 1.0, kWh_TimeMultiplier := 3600.0);
   ZONE_1_AMPS : DINT;
   ZONE_1_POWER_CMD : REAL;
   ZONE_1_SELECT_TE : TE_SELECTED_AVE := (IN_SEL_1ST_TE := 1, IN_SEL_2ND_TE := 1, IN_SEL_3RD_TE := 1, IN_SEL_4TH_TE := 1, IN_1ST_TE := 894.0, IN_2ND_TE := 890.0, IN_3RD_TE := 895.0, IN_4TH_TE := 889.0, OUT_ZONE_1_AVE := 892.0);
   ZONE_1_TEMP_AVE : DINT := 892;
   ZONE_2_AMPS : DINT;
   ZONE_2_POWER_CMD : REAL;
   ZONE_2_SELECT_TE : TE_SELECTED_AVE := (IN_SEL_1ST_TE := 1, IN_SEL_2ND_TE := 1, IN_SEL_3RD_TE := 1, IN_SEL_4TH_TE := 1, IN_1ST_TE := 1171.0, IN_2ND_TE := 1168.0, IN_3RD_TE := 1164.0, IN_4TH_TE := 1156.0, OUT_ZONE_1_AVE := 1164.75);
   ZONE_2_TEMP_AVE : REAL := 1164.75;
   ZONE_3_AMPS : DINT := 7;
   ZONE_3_POWER_CMD : REAL := 3.278298;
   ZONE_3_SELECT_TE : TE_SELECTED_AVE := (IN_SEL_1ST_TE := 1, IN_SEL_2ND_TE := 1, IN_SEL_3RD_TE := 1, IN_SEL_4TH_TE := 1, IN_1ST_TE := 1113.0, IN_2ND_TE := 1108.0, IN_3RD_TE := 1099.0, IN_4TH_TE := 1081.0, OUT_ZONE_1_AVE := 1100.25);
   ZONE_3_TEMP_AVE : REAL := 1100.25;
   ZONE_4_AMPS : DINT;
   ZONE_4_POWER_CMD : REAL;
   ZONE_4_SELECT_TE : TE_SELECTED_AVE := (IN_SEL_1ST_TE := 1, IN_SEL_2ND_TE := 1, IN_SEL_3RD_TE := 1, IN_1ST_TE := 939.0, IN_2ND_TE := 923.0, IN_3RD_TE := 952.0, OUT_ZONE_1_AVE := 938.0);
   ZONE_4_TEMP_AVE : REAL := 938.0;
   ZONE_5_AMPS : DINT;
   ZONE_5_POWER_CMD : REAL;
   ZONE_5_SELECT_TE : TE_SELECTED_AVE := (IN_SEL_1ST_TE := 1, IN_SEL_2ND_TE := 1, IN_SEL_3RD_TE := 1, IN_1ST_TE := 912.0, IN_2ND_TE := 895.0, IN_3RD_TE := 922.0, OUT_ZONE_1_AVE := 909.6667);
   ZONE_5_TEMP_AVE : REAL := 909.6667;
   ZONE_6_AMPS : DINT;
   ZONE_6_POWER_CMD : REAL;
   ZONE_6_SELECT_TE : TE_SELECTED_AVE := (IN_SEL_1ST_TE := 1, IN_SEL_2ND_TE := 1, IN_SEL_3RD_TE := 1, IN_1ST_TE := 1124.0, IN_2ND_TE := 1090.0, IN_3RD_TE := 1096.0, OUT_ZONE_1_AVE := 1103.3334);
   ZONE_6_TEMP_AVE : REAL := 1103.3334;
   ZONE_7_AMPS : DINT;
   ZONE_7_POWER_CMD : REAL;
   ZONE_7_SELECT_TE : TE_SELECTED_AVE := (IN_SEL_1ST_TE := 1, IN_SEL_2ND_TE := 1, IN_SEL_3RD_TE := 1, IN_1ST_TE := 1076.0, IN_2ND_TE := 1093.0, IN_3RD_TE := 1087.0, OUT_ZONE_1_AVE := 1085.3334);
   ZONE_7_TEMP_AVE : REAL := 1085.3334;
   ZONE_8_AMPS : DINT := 19;
   ZONE_8_POWER_CMD : REAL := 17.512012;
   ZONE_8_SELECT_TE : TE_SELECTED_AVE := (IN_SEL_1ST_TE := 1, IN_SEL_2ND_TE := 1, IN_SEL_3RD_TE := 1, IN_1ST_TE := 1101.0, IN_2ND_TE := 1107.0, IN_3RD_TE := 1092.0, OUT_ZONE_1_AVE := 1100.0);
   ZONE_8_TEMP_AVE : REAL := 1100.0;
   ZONE_9_AMPS : DINT := 19;
   ZONE_9_POWER_CMD : REAL := 22.324482;
   ZONE_9_SELECT_TE : TE_SELECTED_AVE := (IN_SEL_1ST_TE := 1, IN_SEL_2ND_TE := 1, IN_SEL_3RD_TE := 1, IN_1ST_TE := 1104.0, IN_2ND_TE := 1093.0, IN_3RD_TE := 1103.0, OUT_ZONE_1_AVE := 1100.0);
   ZONE_9_TEMP_AVE : REAL := 1100.0;
END_VAR

PROGRAM MainProgram   (* main routine MainRoutine *)

ROUTINE A00_SerializeMe   (* ladder *)
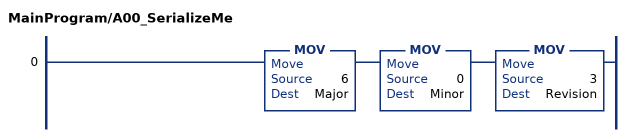
   0: MOV(6,Major)MOV(0,Minor)MOV(3,Revision);
END_ROUTINE

ROUTINE A02_DRYER_MIX_CYCLE   (* ladder *)
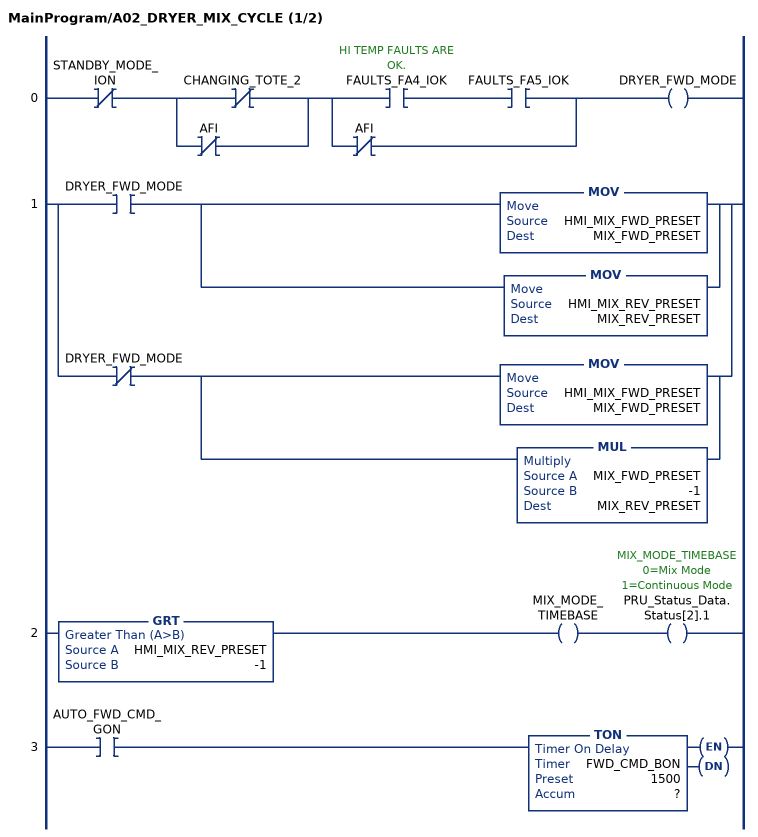
   0: XIO(STANDBY_MODE_ION)[XIO(CHANGING_TOTE_2) ,XIO(AFI) ][XIC(FAULTS_FA4_IOK) XIC(FAULTS_FA5_IOK) ,XIO(AFI) ]OTE(DRYER_FWD_MODE);
   1: [XIC(DRYER_FWD_MODE) [MOV(HMI_MIX_FWD_PRESET,MIX_FWD_PRESET) ,MOV(HMI_MIX_REV_PRESET,MIX_REV_PRESET) ] ,XIO(DRYER_FWD_MODE) [MOV(HMI_MIX_FWD_PRESET,MIX_FWD_PRESET) ,MUL(MIX_FWD_PRESET,-1,MIX_REV_PRESET) ] ];
   2: GRT(HMI_MIX_REV_PRESET,-1)OTE(MIX_MODE_TIMEBASE)OTE(PRU_Status_Data.Status[2].1);
   3: XIC(AUTO_FWD_CMD_GON)TON(FWD_CMD_BON,?,?);
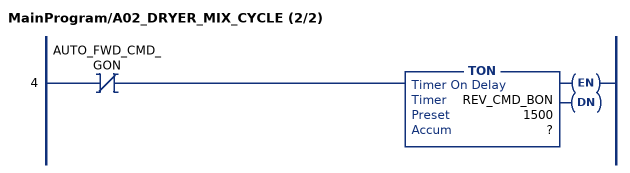
   4: XIO(AUTO_FWD_CMD_GON)TON(REV_CMD_BON,?,?);
END_ROUTINE

ROUTINE A04_KG021_CONTROL   (* ladder *)
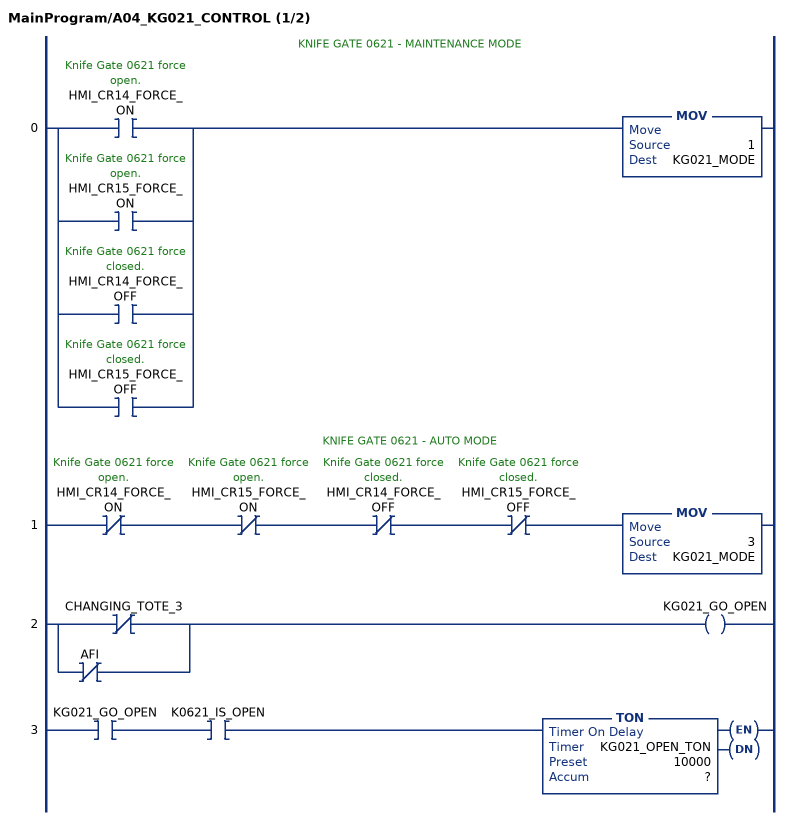
   // KNIFE GATE 0621 - MAINTENANCE MODE
   0: [XIC(HMI_CR14_FORCE_ON) ,XIC(HMI_CR15_FORCE_ON) ,XIC(HMI_CR14_FORCE_OFF) ,XIC(HMI_CR15_FORCE_OFF) ]MOV(1,KG021_MODE);
   // KNIFE GATE 0621 - AUTO MODE
   1: XIO(HMI_CR14_FORCE_ON)XIO(HMI_CR15_FORCE_ON)XIO(HMI_CR14_FORCE_OFF)XIO(HMI_CR15_FORCE_OFF)MOV(3,KG021_MODE);
   2: [XIO(CHANGING_TOTE_3) ,XIO(AFI) ]OTE(KG021_GO_OPEN);
   3: XIC(KG021_GO_OPEN)XIC(K0621_IS_OPEN)TON(KG021_OPEN_TON,?,?);
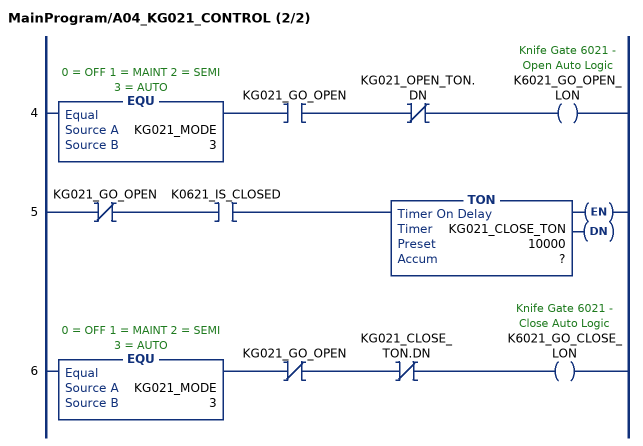
   4: EQU(KG021_MODE,3)XIC(KG021_GO_OPEN)XIO(KG021_OPEN_TON.DN)OTE(K6021_GO_OPEN_LON);
   5: XIO(KG021_GO_OPEN)XIC(K0621_IS_CLOSED)TON(KG021_CLOSE_TON,?,?);
   6: EQU(KG021_MODE,3)XIO(KG021_GO_OPEN)XIO(KG021_CLOSE_TON.DN)OTE(K6021_GO_CLOSE_LON);
END_ROUTINE

ROUTINE A05_COOLSCREW_CONTROL   (* ladder *)
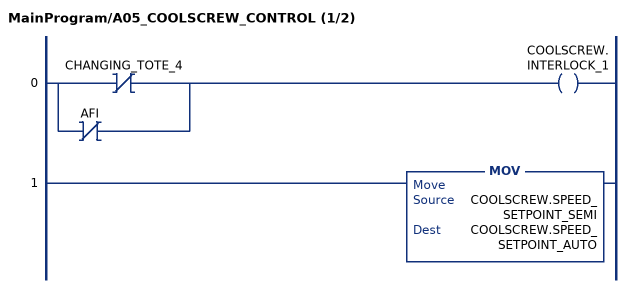
   0: [XIO(CHANGING_TOTE_4) ,XIO(AFI) ]OTE(COOLSCREW.INTERLOCK_1);
   1: MOV(COOLSCREW.SPEED_SETPOINT_SEMI,COOLSCREW.SPEED_SETPOINT_AUTO);
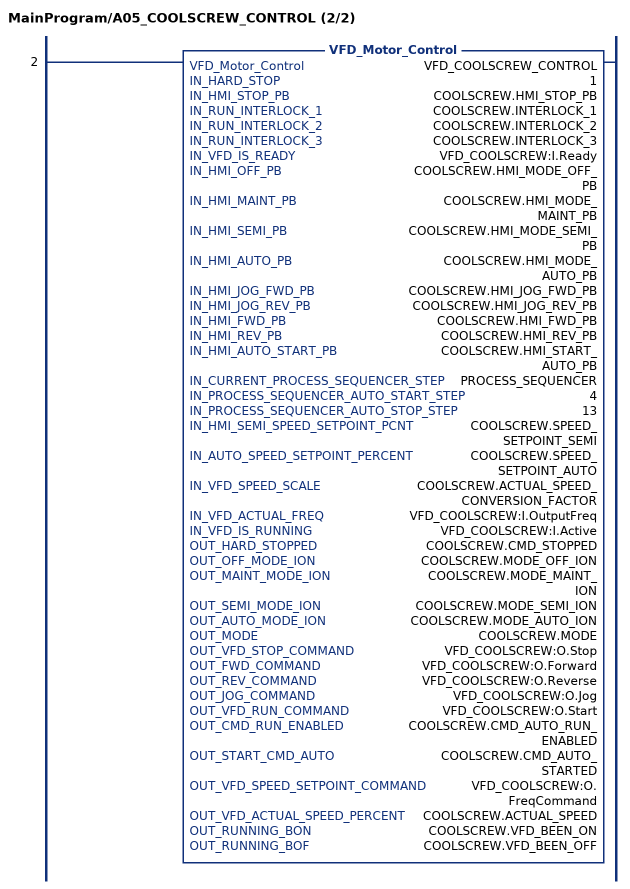
   2: VFD_Motor_Control(VFD_COOLSCREW_CONTROL,1,COOLSCREW.HMI_STOP_PB,COOLSCREW.INTERLOCK_1,COOLSCREW.INTERLOCK_2,COOLSCREW.INTERLOCK_3,VFD_COOLSCREW:I.Ready,COOLSCREW.HMI_MODE_OFF_PB,COOLSCREW.HMI_MODE_MAINT_PB,COOLSCREW.HMI_MODE_SEMI_PB,COOLSCREW.HMI_MODE_AUTO_PB,COOLSCREW.HMI_JOG_FWD_PB,COOLSCREW.HMI_JOG_REV_PB,COOLSCREW.HMI_FWD_PB,COOLSCREW.HMI_REV_PB,COOLSCREW.HMI_START_AUTO_PB,PROCESS_SEQUENCER,4,13,COOLSCREW.SPEED_SETPOINT_SEMI,COOLSCREW.SPEED_SETPOINT_AUTO,COOLSCREW.ACTUAL_SPEED_CONVERSION_FACTOR,VFD_COOLSCREW:I.OutputFreq,VFD_COOLSCREW:I.Active,COOLSCREW.CMD_STOPPED,COOLSCREW.MODE_OFF_ION,COOLSCREW.MODE_MAINT_ION,COOLSCREW.MODE_SEMI_ION,COOLSCREW.MODE_AUTO_ION,COOLSCREW.MODE,VFD_COOLSCREW:O.Stop,VFD_COOLSCREW:O.Forward,VFD_COOLSCREW:O.Reverse,VFD_COOLSCREW:O.Jog,VFD_COOLSCREW:O.Start,COOLSCREW.CMD_AUTO_RUN_ENABLED,COOLSCREW.CMD_AUTO_STARTED,VFD_COOLSCREW:O.FreqCommand,COOLSCREW.ACTUAL_SPEED,COOLSCREW.VFD_BEEN_ON,COOLSCREW.VFD_BEEN_OFF);
END_ROUTINE

ROUTINE A06_KG022_CONTROL   (* ladder *)
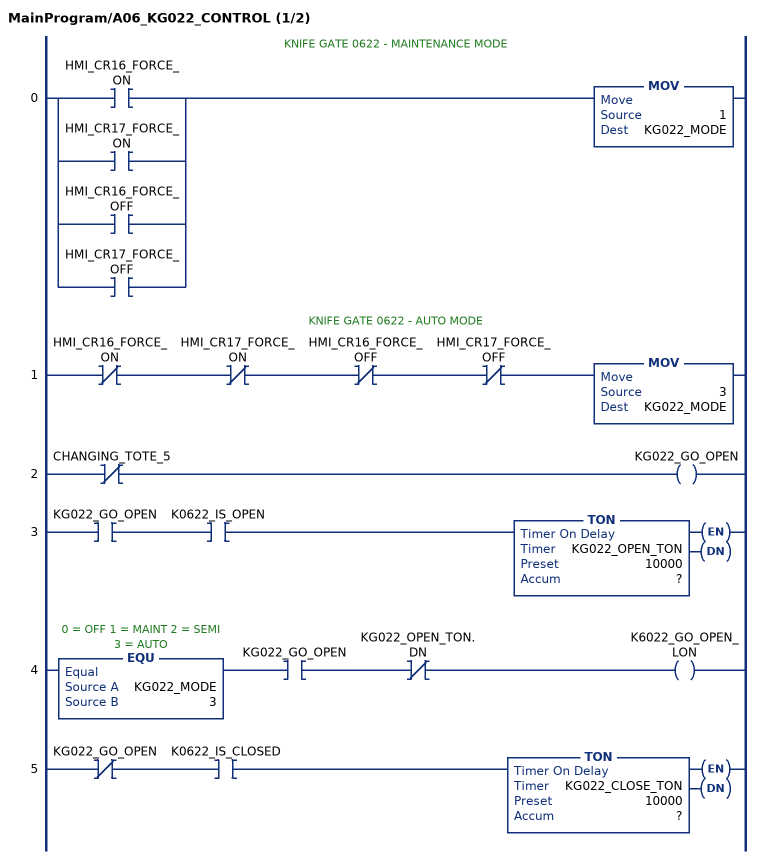
   // KNIFE GATE 0622 - MAINTENANCE MODE
   0: [XIC(HMI_CR16_FORCE_ON) ,XIC(HMI_CR17_FORCE_ON) ,XIC(HMI_CR16_FORCE_OFF) ,XIC(HMI_CR17_FORCE_OFF) ]MOV(1,KG022_MODE);
   // KNIFE GATE 0622 - AUTO MODE
   1: XIO(HMI_CR16_FORCE_ON)XIO(HMI_CR17_FORCE_ON)XIO(HMI_CR16_FORCE_OFF)XIO(HMI_CR17_FORCE_OFF)MOV(3,KG022_MODE);
   2: XIO(CHANGING_TOTE_5)OTE(KG022_GO_OPEN);
   3: XIC(KG022_GO_OPEN)XIC(K0622_IS_OPEN)TON(KG022_OPEN_TON,?,?);
   4: EQU(KG022_MODE,3)XIC(KG022_GO_OPEN)XIO(KG022_OPEN_TON.DN)OTE(K6022_GO_OPEN_LON);
   5: XIO(KG022_GO_OPEN)XIC(K0622_IS_CLOSED)TON(KG022_CLOSE_TON,?,?);
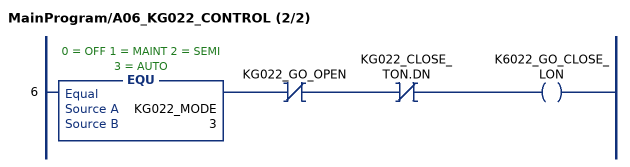
   6: EQU(KG022_MODE,3)XIO(KG022_GO_OPEN)XIO(KG022_CLOSE_TON.DN)OTE(K6022_GO_CLOSE_LON);
END_ROUTINE
